LIN {X 0,Y 530.945,Z 338.971,A -85,B 0,C 180,E1 -4197.132,E2 -4197.132} C_VEL
LIN {X 0,Y 530.932,Z 338.967,A -85,B 0,C 180,E1 -4199.801,E2 -4199.801} C_VEL
LIN {X 0,Y 530.986,Z 339.128,A -85,B 0,C 180,E1 -4201.443,E2 -4201.443} C_VEL
LIN {X 0,Y 533.881,Z 351.837,A -85,B 0,C 180,E1 -4203.201,E2 -4203.201} C_VEL
LIN {X 0,Y 533.349,Z 375.523,A -85,B 0,C 180,E1 -4206.096,E2 -4206.096} C_VEL
LIN {X 0,Y 532.844,Z 398.324,A -85,B 0,C 180,E1 -4208.824,E2 -4208.824} C_VEL
LIN {X 0,Y 535.193,Z 410.616,A -85,B 0,C 180,E1 -4209.118,E2 -4209.118} C_VEL
LIN {X 0,Y 534.278,Z 564.153,A -85,B 0,C 180,E1 -4211.249,E2 -4211.249} C_VEL
LIN {X 0,Y 534.01,Z 579.764,A -85,B 0,C 180,E1 -4211.612,E2 -4211.612} C_VEL
LIN {X 0,Y 533.688,Z 594.764,A -85,B 0,C 180,E1 -4212.122,E2 -4212.122} C_VEL
LIN {X 0,Y 533.332,Z 608.76,A -85,B 0,C 180,E1 -4212.753,E2 -4212.753} C_VEL
LIN {X 0,Y 532.844,Z 622.489,A -85,B 0,C 180,E1 -4213.526,E2 -4213.526} C_VEL
LIN {X 0,Y 532.401,Z 636.442,A -85,B 0,C 180,E1 -4214.503,E2 -4214.503} C_VEL
LIN {X 0,Y 531.99,Z 647.758,A -85,B 0,C 180,E1 -4215.463,E2 -4215.463} C_VEL
LIN {X 0,Y 531.655,Z 657.488,A -85,B 0,C 180,E1 -4216.43,E2 -4216.43} C_VEL
LIN {X 0,Y 531.343,Z 665.917,A -85,B 0,C 180,E1 -4217.394,E2 -4217.394} C_VEL
LIN {X 0,Y 531.108,Z 672.885,A -85,B 0,C 180,E1 -4218.3,E2 -4218.3} C_VEL
LIN {X 0,Y 531.005,Z 679.757,A -85,B 0,C 180,E1 -4219.322,E2 -4219.322} C_VEL
LIN {X 0,Y 530.768,Z 686.452,A -85,B 0,C 180,E1 -4220.473,E2 -4220.473} C_VEL
LIN {X 0,Y 530.667,Z 692.162,A -85,B 0,C 180,E1 -4221.623,E2 -4221.623} C_VEL
LIN {X 0,Y 530.573,Z 696.984,A -85,B 0,C 180,E1 -4222.771,E2 -4222.771} C_VEL
LIN {X 0,Y 530.515,Z 701.005,A -85,B 0,C 180,E1 -4223.916,E2 -4223.916} C_VEL
LIN {X 0,Y 530.412,Z 705.143,A -85,B 0,C 180,E1 -4225.44,E2 -4225.44} C_VEL
LIN {X 0,Y 530.481,Z 706.833,A -85,B 0,C 180,E1 -4226.202,E2 -4226.202} C_VEL
LIN {X 0,Y 530.409,Z 709.125,A -85,B 0,C 180,E1 -4227.722,E2 -4227.722} C_VEL
LIN {X 0,Y 530.34,Z 710.269,A -85,B 0,C 180,E1 -4229.241,E2 -4229.241} C_VEL
LIN {X 0,Y 530.341,Z 710.497,A -85,B 0,C 180,E1 -4230,E2 -4230} C_VEL
LIN {X 0,Y 530.359,Z 709.942,A -85,B 0,C 180,E1 -4231.519,E2 -4231.519} C_VEL
LIN {X 0,Y 530.45,Z 708.224,A -85,B 0,C 180,E1 -4233.038,E2 -4233.038} C_VEL
LIN {X 0,Y 530.481,Z 706.999,A -85,B 0,C 180,E1 -4233.798,E2 -4233.798} C_VEL
LIN {X 0,Y 530.508,Z 703.526,A -85,B 0,C 180,E1 -4235.321,E2 -4235.321} C_VEL
LIN {X 0,Y 530.55,Z 698.716,A -85,B 0,C 180,E1 -4236.847,E2 -4236.847} C_VEL
LIN {X 0,Y 530.636,Z 694.25,A -85,B 0,C 180,E1 -4237.994,E2 -4237.994} C_VEL
LIN {X 0,Y 530.742,Z 688.921,A -85,B 0,C 180,E1 -4239.143,E2 -4239.143} C_VEL
LIN {X 0,Y 530.926,Z 682.638,A -85,B 0,C 180,E1 -4240.294,E2 -4240.294} C_VEL
LIN {X 0,Y 531.066,Z 675.267,A -85,B 0,C 180,E1 -4241.45,E2 -4241.45} C_VEL
LIN {X 0,Y 531.288,Z 668.195,A -85,B 0,C 180,E1 -4242.413,E2 -4242.413} C_VEL
LIN {X 0,Y 531.589,Z 660.096,A -85,B 0,C 180,E1 -4243.377,E2 -4243.377} C_VEL
LIN {X 0,Y 531.893,Z 650.752,A -85,B 0,C 180,E1 -4244.344,E2 -4244.344} C_VEL
LIN {X 0,Y 532.284,Z 639.846,A -85,B 0,C 180,E1 -4245.312,E2 -4245.312} C_VEL
LIN {X 0,Y 532.646,Z 628.232,A -85,B 0,C 180,E1 -4246.185,E2 -4246.185} C_VEL
LIN {X 0,Y 533.167,Z 614.163,A -85,B 0,C 180,E1 -4247.055,E2 -4247.055} C_VEL
LIN {X 0,Y 533.547,Z 600.41,A -85,B 0,C 180,E1 -4247.734,E2 -4247.734} C_VEL
LIN {X 0,Y 533.892,Z 585.818,A -85,B 0,C 180,E1 -4248.293,E2 -4248.293} C_VEL
LIN {X 0,Y 534.167,Z 571.375,A -85,B 0,C 180,E1 -4248.694,E2 -4248.694} C_VEL
LIN {X 0,Y 534.375,Z 554.599,A -85,B 0,C 180,E1 -4248.991,E2 -4248.991} C_VEL
LIN {X 0,Y 535.195,Z 410.641,A -85,B 0,C 180,E1 -4250.972,E2 -4250.972} C_VEL
LIN {X 0,Y 532.855,Z 398.387,A -85,B 0,C 180,E1 -4251.256,E2 -4251.256} C_VEL
LIN {X 0,Y 533.401,Z 372.991,A -85,B 0,C 180,E1 -4254.303,E2 -4254.303} C_VEL
LIN {X 0,Y 533.864,Z 352.576,A -85,B 0,C 180,E1 -4256.8,E2 -4256.8} C_VEL
LIN {X 0,Y 533.375,Z 349.148,A -85,B 0,C 180,E1 -4257.25,E2 -4257.25} C_VEL
LIN {X 0,Y 530.957,Z 339.096,A -85,B 0,C 180,E1 -4258.66,E2 -4258.66} C_VEL
LIN {X 0,Y 530.935,Z 338.972,A -85,B 0,C 180,E1 -4261.081,E2 -4261.081} C_VEL
LIN {X 0,Y 530.932,Z 338.973,A -85,B 0,C 180,E1 -4263.777,E2 -4263.777} C_VEL
LIN {X 0,Y 530.902,Z 338.976,A -85,B 0,C 180,E1 -4266.563,E2 -4266.563} C_VEL
LIN {X 0,Y 530.938,Z 338.971,A -85,B 0,C 180,E1 -4269.448,E2 -4269.448} C_VEL
LIN {X 0,Y 530.91,Z 338.974,A -85,B 0,C 180,E1 -4272.463,E2 -4272.463} C_VEL
LIN {X 0,Y 530.963,Z 338.969,A -85,B 0,C 180,E1 -4275.45,E2 -4275.45} C_VEL
LIN {X 0,Y 530.918,Z 338.973,A -85,B 0,C 180,E1 -4278.557,E2 -4278.557} C_VEL
LIN {X 0,Y 530.947,Z 338.972,A -85,B 0,C 180,E1 -4281.528,E2 -4281.528} C_VEL
LIN {X 0,Y 530.934,Z 338.969,A -85,B 0,C 180,E1 -4284.378,E2 -4284.378} C_VEL
LIN {X 0,Y 530.967,Z 338.967,A -85,B 0,C 180,E1 -4287.133,E2 -4287.133} C_VEL
LIN {X 0,Y 530.96,Z 338.975,A -85,B 0,C 180,E1 -4289.802,E2 -4289.802} C_VEL
LIN {X 0,Y 530.963,Z 338.963,A -85,B 0,C 180,E1 -4292.478,E2 -4292.478} C_VEL
LIN {X 0,Y 530.95,Z 338.968,A -85,B 0,C 180,E1 -4294.94,E2 -4294.94} C_VEL
LIN {X 0,Y 530.978,Z 338.967,A -85,B 0,C 180,E1 -4297.898,E2 -4297.898} C_VEL
LIN {X 0,Y 530.983,Z 338.964,A -85,B 0,C 180,E1 -4300.677,E2 -4300.677} C_VEL
LIN {X 0,Y 530.965,Z 338.965,A -85,B 0,C 180,E1 -4303.07,E2 -4303.07} C_VEL
LIN {X 0,Y 531.02,Z 338.965,A -85,B 0,C 180,E1 -4305.436,E2 -4305.436} C_VEL
LIN {X 0,Y 531.036,Z 338.953,A -85,B 0,C 180,E1 -4308.55,E2 -4308.55} C_VEL
LIN {X 0,Y 531.035,Z 338.965,A -85,B 0,C 180,E1 -4311.629,E2 -4311.629} C_VEL
LIN {X 0,Y 531.117,Z 338.943,A -85,B 0,C 180,E1 -4314.685,E2 -4314.685} C_VEL
LIN {X 0,Y 531.14,Z 338.949,A -85,B 0,C 180,E1 -4317.725,E2 -4317.725} C_VEL
LIN {X 0,Y 531.149,Z 338.941,A -85,B 0,C 180,E1 -4320.758,E2 -4320.758} C_VEL
LIN {X 0,Y 531.101,Z 338.949,A -85,B 0,C 180,E1 -4323.034,E2 -4323.034} C_VEL
LIN {X 0,Y 531.074,Z 338.951,A -85,B 0,C 180,E1 -4326.077,E2 -4326.077} C_VEL
LIN {X 0,Y 531.023,Z 338.96,A -85,B 0,C 180,E1 -4329.138,E2 -4329.138} C_VEL
LIN {X 0,Y 531.041,Z 338.954,A -85,B 0,C 180,E1 -4332.225,E2 -4332.225} C_VEL
LIN {X 0,Y 530.994,Z 338.968,A -85,B 0,C 180,E1 -4335.35,E2 -4335.35} C_VEL
LIN {X 0,Y 530.987,Z 338.962,A -85,B 0,C 180,E1 -4338.521,E2 -4338.521} C_VEL
LIN {X 0,Y 530.999,Z 338.963,A -85,B 0,C 180,E1 -4340.938,E2 -4340.938} C_VEL
LIN {X 0,Y 530.966,Z 338.963,A -85,B 0,C 180,E1 -4344.225,E2 -4344.225} C_VEL
LIN {X 0,Y 531.002,Z 338.963,A -85,B 0,C 180,E1 -4346.744,E2 -4346.744} C_VEL
LIN {X 0,Y 530.982,Z 338.966,A -85,B 0,C 180,E1 -4349.322,E2 -4349.322} C_VEL
LIN {X 0,Y 530.966,Z 338.966,A -85,B 0,C 180,E1 -4352.1,E2 -4352.1} C_VEL
LIN {X 0,Y 530.97,Z 338.968,A -85,B 0,C 180,E1 -4354.851,E2 -4354.851} C_VEL
LIN {X 0,Y 530.966,Z 338.967,A -85,B 0,C 180,E1 -4357.508,E2 -4357.508} C_VEL
LIN {X 0,Y 530.984,Z 338.952,A -85,B 0,C 180,E1 -4360.433,E2 -4360.433} C_VEL
LIN {X 0,Y 530.965,Z 338.969,A -85,B 0,C 180,E1 -4363.494,E2 -4363.494} C_VEL
LIN {X 0,Y 530.965,Z 338.963,A -85,B 0,C 180,E1 -4366.505,E2 -4366.505} C_VEL
LIN {X 0,Y 530.985,Z 338.965,A -85,B 0,C 180,E1 -4369.567,E2 -4369.567} C_VEL
LIN {X 0,Y 530.968,Z 338.971,A -85,B 0,C 180,E1 -4372.577,E2 -4372.577} C_VEL
LIN {X 0,Y 530.982,Z 338.969,A -85,B 0,C 180,E1 -4375.31,E2 -4375.31} C_VEL
LIN {X 0,Y 530.968,Z 338.967,A -85,B 0,C 180,E1 -4378.032,E2 -4378.032} C_VEL
LIN {X 0,Y 530.989,Z 338.971,A -85,B 0,C 180,E1 -4380.874,E2 -4380.874} C_VEL
LIN {X 0,Y 531.044,Z 339.142,A -85,B 0,C 180,E1 -4381.924,E2 -4381.924} C_VEL
LIN {X 0,Y 534.398,Z 352.329,A -85,B 0,C 180,E1 -4383.691,E2 -4383.691} C_VEL
LIN {X 0,Y 533.668,Z 375.374,A -85,B 0,C 180,E1 -4386.318,E2 -4386.318} C_VEL
LIN {X 0,Y 533.029,Z 397.899,A -85,B 0,C 180,E1 -4388.826,E2 -4388.826} C_VEL
LIN {X 0,Y 535.1,Z 409.701,A -85,B 0,C 180,E1 -4389.1,E2 -4389.1} C_VEL
LIN {X 0,Y 534.127,Z 564.616,A -85,B 0,C 180,E1 -4391.261,E2 -4391.261} C_VEL
LIN {X 0,Y 533.892,Z 580.328,A -85,B 0,C 180,E1 -4391.633,E2 -4391.633} C_VEL
LIN {X 0,Y 533.573,Z 594.596,A -85,B 0,C 180,E1 -4392.118,E2 -4392.118} C_VEL
LIN {X 0,Y 533.2,Z 608.743,A -85,B 0,C 180,E1 -4392.749,E2 -4392.749} C_VEL
LIN {X 0,Y 532.766,Z 622.554,A -85,B 0,C 180,E1 -4393.524,E2 -4393.524} C_VEL
LIN {X 0,Y 532.379,Z 635.728,A -85,B 0,C 180,E1 -4394.434,E2 -4394.434} C_VEL
LIN {X 0,Y 531.954,Z 648.089,A -85,B 0,C 180,E1 -4395.462,E2 -4395.462} C_VEL
LIN {X 0,Y 531.608,Z 659.731,A -85,B 0,C 180,E1 -4396.623,E2 -4396.623} C_VEL
LIN {X 0,Y 531.286,Z 669.388,A -85,B 0,C 180,E1 -4397.781,E2 -4397.781} C_VEL
LIN {X 0,Y 531.051,Z 678.853,A -85,B 0,C 180,E1 -4399.13,E2 -4399.13} C_VEL
LIN {X 0,Y 530.764,Z 686.735,A -85,B 0,C 180,E1 -4400.473,E2 -4400.473} C_VEL
LIN {X 0,Y 530.64,Z 694.089,A -85,B 0,C 180,E1 -4402.006,E2 -4402.006} C_VEL
LIN {X 0,Y 530.545,Z 699.699,A -85,B 0,C 180,E1 -4403.467,E2 -4403.467} C_VEL
LIN {X 0,Y 530.509,Z 703.386,A -85,B 0,C 180,E1 -4404.679,E2 -4404.679} C_VEL
LIN {X 0,Y 530.481,Z 706.887,A -85,B 0,C 180,E1 -4406.202,E2 -4406.202} C_VEL
LIN {X 0,Y 530.408,Z 709.189,A -85,B 0,C 180,E1 -4407.722,E2 -4407.722} C_VEL
LIN {X 0,Y 530.34,Z 710.348,A -85,B 0,C 180,E1 -4409.241,E2 -4409.241} C_VEL
LIN {X 0,Y 530.34,Z 710.347,A -85,B 0,C 180,E1 -4410.759,E2 -4410.759} C_VEL
LIN {X 0,Y 530.408,Z 709.185,A -85,B 0,C 180,E1 -4412.278,E2 -4412.278} C_VEL
LIN {X 0,Y 530.481,Z 706.882,A -85,B 0,C 180,E1 -4413.798,E2 -4413.798} C_VEL
LIN {X 0,Y 530.509,Z 703.386,A -85,B 0,C 180,E1 -4415.321,E2 -4415.321} C_VEL
LIN {X 0,Y 530.55,Z 698.609,A -85,B 0,C 180,E1 -4416.847,E2 -4416.847} C_VEL
LIN {X 0,Y 530.665,Z 692.419,A -85,B 0,C 180,E1 -4418.377,E2 -4418.377} C_VEL
LIN {X 0,Y 530.809,Z 684.641,A -85,B 0,C 180,E1 -4419.911,E2 -4419.911} C_VEL
LIN {X 0,Y 531.056,Z 676.365,A -85,B 0,C 180,E1 -4421.257,E2 -4421.257} C_VEL
LIN {X 0,Y 531.383,Z 666.39,A -85,B 0,C 180,E1 -4422.605,E2 -4422.605} C_VEL
LIN {X 0,Y 531.708,Z 656.119,A -85,B 0,C 180,E1 -4423.764,E2 -4423.764} C_VEL
LIN {X 0,Y 532.084,Z 643.687,A -85,B 0,C 180,E1 -4424.926,E2 -4424.926} C_VEL
LIN {X 0,Y 532.515,Z 631.406,A -85,B 0,C 180,E1 -4425.877,E2 -4425.877} C_VEL
LIN {X 0,Y 532.924,Z 617.492,A -85,B 0,C 180,E1 -4426.767,E2 -4426.767} C_VEL
LIN {X 0,Y 533.287,Z 603.31,A -85,B 0,C 180,E1 -4427.496,E2 -4427.496} C_VEL
LIN {X 0,Y 533.618,Z 588.738,A -85,B 0,C 180,E1 -4428.079,E2 -4428.079} C_VEL
LIN {X 0,Y 533.959,Z 573.588,A -85,B 0,C 180,E1 -4428.522,E2 -4428.522} C_VEL
LIN {X 0,Y 534.141,Z 557.458,A -85,B 0,C 180,E1 -4428.83,E2 -4428.83} C_VEL
LIN {X 0,Y 534.954,Z 409.306,A -85,B 0,C 180,E1 -4430.883,E2 -4430.883} C_VEL
LIN {X 0,Y 533.023,Z 398.201,A -85,B 0,C 180,E1 -4431.125,E2 -4431.125} C_VEL
LIN {X 0,Y 533.541,Z 376.812,A -85,B 0,C 180,E1 -4433.482,E2 -4433.482} C_VEL
LIN {X 0,Y 534.319,Z 352.2,A -85,B 0,C 180,E1 -4436.292,E2 -4436.292} C_VEL
LIN {X 0,Y 531.049,Z 339.118,A -85,B 0,C 180,E1 -4438.089,E2 -4438.089} C_VEL
LIN {X 0,Y 530.958,Z 338.975,A -85,B 0,C 180,E1 -4441.079,E2 -4441.079} C_VEL
LIN {X 0,Y 530.99,Z 338.965,A -85,B 0,C 180,E1 -4443.773,E2 -4443.773} C_VEL
LIN {X 0,Y 530.96,Z 338.974,A -85,B 0,C 180,E1 -4446.558,E2 -4446.558} C_VEL
LIN {X 0,Y 530.987,Z 338.967,A -85,B 0,C 180,E1 -4449.444,E2 -4449.444} C_VEL
LIN {X 0,Y 530.979,Z 338.971,A -85,B 0,C 180,E1 -4452.457,E2 -4452.457} C_VEL
LIN {X 0,Y 530.978,Z 338.967,A -85,B 0,C 180,E1 -4455.622,E2 -4455.622} C_VEL
LIN {X 0,Y 530.99,Z 338.972,A -85,B 0,C 180,E1 -4458.564,E2 -4458.564} C_VEL
LIN {X 0,Y 530.954,Z 338.97,A -85,B 0,C 180,E1 -4461.529,E2 -4461.529} C_VEL
LIN {X 0,Y 530.948,Z 338.977,A -85,B 0,C 180,E1 -4464.38,E2 -4464.38} C_VEL
LIN {X 0,Y 530.967,Z 338.97,A -85,B 0,C 180,E1 -4467.133,E2 -4467.133} C_VEL
LIN {X 0,Y 530.948,Z 338.975,A -85,B 0,C 180,E1 -4469.802,E2 -4469.802} C_VEL
LIN {X 0,Y 530.954,Z 338.976,A -85,B 0,C 180,E1 -4472.48,E2 -4472.48} C_VEL
LIN {X 0,Y 530.993,Z 339.163,A -85,B 0,C 180,E1 -4473.442,E2 -4473.442} C_VEL
LIN {X 0,Y 533.281,Z 349.071,A -85,B 0,C 180,E1 -4475.057,E2 -4475.057} C_VEL
LIN {X 0,Y 533.456,Z 353.457,A -85,B 0,C 180,E1 -4475.699,E2 -4475.699} C_VEL
LIN {X 0,Y 532.723,Z 376.404,A -85,B 0,C 180,E1 -4478.931,E2 -4478.931} C_VEL
LIN {X 0,Y 532.137,Z 397.45,A -85,B 0,C 180,E1 -4481.828,E2 -4481.828} C_VEL
LIN {X 0,Y 533.286,Z 403.741,A -85,B 0,C 180,E1 -4482.001,E2 -4482.001} C_VEL
LIN {X 0,Y 534.066,Z 408.919,A -85,B 0,C 180,E1 -4482.11,E2 -4482.11} C_VEL
LIN {X 0,Y 533.219,Z 536.961,A -85,B 0,C 180,E1 -4483.949,E2 -4483.949} C_VEL
LIN {X 0,Y 532.942,Z 551.427,A -85,B 0,C 180,E1 -4484.314,E2 -4484.314} C_VEL
LIN {X 0,Y 532.714,Z 565.736,A -85,B 0,C 180,E1 -4484.848,E2 -4484.848} C_VEL
LIN {X 0,Y 532.412,Z 578.426,A -85,B 0,C 180,E1 -4485.475,E2 -4485.475} C_VEL
LIN {X 0,Y 532.053,Z 590.85,A -85,B 0,C 180,E1 -4486.245,E2 -4486.245} C_VEL
LIN {X 0,Y 531.733,Z 602.123,A -85,B 0,C 180,E1 -4487.112,E2 -4487.112} C_VEL
LIN {X 0,Y 531.422,Z 613.157,A -85,B 0,C 180,E1 -4488.138,E2 -4488.138} C_VEL
LIN {X 0,Y 531.208,Z 622,A -85,B 0,C 180,E1 -4489.133,E2 -4489.133} C_VEL
LIN {X 0,Y 530.929,Z 630.682,A -85,B 0,C 180,E1 -4490.284,E2 -4490.284} C_VEL
LIN {X 0,Y 530.743,Z 638.877,A -85,B 0,C 180,E1 -4491.625,E2 -4491.625} C_VEL
LIN {X 0,Y 530.587,Z 644.644,A -85,B 0,C 180,E1 -4492.771,E2 -4492.771} C_VEL
LIN {X 0,Y 530.566,Z 650.752,A -85,B 0,C 180,E1 -4494.299,E2 -4494.299} C_VEL
LIN {X 0,Y 530.449,Z 654.284,A -85,B 0,C 180,E1 -4495.441,E2 -4495.441} C_VEL
LIN {X 0,Y 530.453,Z 657.771,A -85,B 0,C 180,E1 -4496.962,E2 -4496.962} C_VEL
LIN {X 0,Y 530.359,Z 659.74,A -85,B 0,C 180,E1 -4498.481,E2 -4498.481} C_VEL
LIN {X 0,Y 530.342,Z 660.496,A -85,B 0,C 180,E1 -4500,E2 -4500} C_VEL
LIN {X 0,Y 530.357,Z 659.816,A -85,B 0,C 180,E1 -4501.519,E2 -4501.519} C_VEL
LIN {X 0,Y 530.452,Z 657.919,A -85,B 0,C 180,E1 -4503.038,E2 -4503.038} C_VEL
LIN {X 0,Y 530.448,Z 654.528,A -85,B 0,C 180,E1 -4504.56,E2 -4504.56} C_VEL
LIN {X 0,Y 530.568,Z 649.767,A -85,B 0,C 180,E1 -4506.083,E2 -4506.083} C_VEL
LIN {X 0,Y 530.64,Z 643.271,A -85,B 0,C 180,E1 -4507.611,E2 -4507.611} C_VEL
LIN {X 0,Y 530.809,Z 636.09,A -85,B 0,C 180,E1 -4508.95,E2 -4508.95} C_VEL
LIN {X 0,Y 530.982,Z 628.546,A -85,B 0,C 180,E1 -4510.101,E2 -4510.101} C_VEL
LIN {X 0,Y 531.274,Z 619.564,A -85,B 0,C 180,E1 -4511.252,E2 -4511.252} C_VEL
LIN {X 0,Y 531.459,Z 610.473,A -85,B 0,C 180,E1 -4512.215,E2 -4512.215} C_VEL
LIN {X 0,Y 531.82,Z 599.737,A -85,B 0,C 180,E1 -4513.177,E2 -4513.177} C_VEL
LIN {X 0,Y 532.121,Z 587.852,A -85,B 0,C 180,E1 -4514.045,E2 -4514.045} C_VEL
LIN {X 0,Y 532.518,Z 574.763,A -85,B 0,C 180,E1 -4514.815,E2 -4514.815} C_VEL
LIN {X 0,Y 532.84,Z 562.962,A -85,B 0,C 180,E1 -4515.36,E2 -4515.36} C_VEL
LIN {X 0,Y 533.045,Z 549.361,A -85,B 0,C 180,E1 -4515.839,E2 -4515.839} C_VEL
LIN {X 0,Y 533.237,Z 536.026,A -85,B 0,C 180,E1 -4516.166,E2 -4516.166} C_VEL
LIN {X 0,Y 533.921,Z 407.703,A -85,B 0,C 180,E1 -4517.973,E2 -4517.973} C_VEL
LIN {X 0,Y 532.113,Z 397.871,A -85,B 0,C 180,E1 -4518.204,E2 -4518.204} C_VEL
LIN {X 0,Y 532.073,Z 396.512,A -85,B 0,C 180,E1 -4518.329,E2 -4518.329} C_VEL
LIN {X 0,Y 532.671,Z 373.671,A -85,B 0,C 180,E1 -4521.477,E2 -4521.477} C_VEL
LIN {X 0,Y 533.099,Z 360.019,A -85,B 0,C 180,E1 -4523.384,E2 -4523.384} C_VEL
LIN {X 0,Y 532.535,Z 356.591,A -85,B 0,C 180,E1 -4523.898,E2 -4523.898} C_VEL
LIN {X 0,Y 530.909,Z 353.505,A -85,B 0,C 180,E1 -4524.419,E2 -4524.419} C_VEL
LIN {X 0,Y 525.491,Z 345.703,A -85,B 0,C 180,E1 -4525.83,E2 -4525.83} C_VEL
LIN {X 0,Y 524.749,Z 343.526,A -85,B 0,C 180,E1 -4526.19,E2 -4526.19} C_VEL
LIN {X 0,Y 523.916,Z 339.972,A -85,B 0,C 180,E1 -4526.812,E2 -4526.812} C_VEL
LIN {X 0,Y 523.868,Z 339.856,A -85,B 0,C 180,E1 -4529.761,E2 -4529.761} C_VEL
LIN {X 0,Y 523.896,Z 339.852,A -85,B 0,C 180,E1 -4532.452,E2 -4532.452} C_VEL
LIN {X 0,Y 523.882,Z 339.85,A -85,B 0,C 180,E1 -4535.23,E2 -4535.23} C_VEL
LIN {X 0,Y 523.888,Z 339.856,A -85,B 0,C 180,E1 -4538.104,E2 -4538.104} C_VEL
LIN {X 0,Y 523.876,Z 339.849,A -85,B 0,C 180,E1 -4541.3,E2 -4541.3} C_VEL
LIN {X 0,Y 523.93,Z 339.845,A -85,B 0,C 180,E1 -4544.688,E2 -4544.688} C_VEL
LIN {X 0,Y 523.886,Z 339.85,A -85,B 0,C 180,E1 -4547.874,E2 -4547.874} C_VEL
LIN {X 0,Y 523.894,Z 339.846,A -85,B 0,C 180,E1 -4551.084,E2 -4551.084} C_VEL
LIN {X 0,Y 523.853,Z 339.855,A -85,B 0,C 180,E1 -4553.821,E2 -4553.821} C_VEL
LIN {X 0,Y 523.896,Z 339.851,A -85,B 0,C 180,E1 -4556.632,E2 -4556.632} C_VEL
LIN {X 0,Y 523.908,Z 339.847,A -85,B 0,C 180,E1 -4559.352,E2 -4559.352} C_VEL
LIN {X 0,Y 523.953,Z 340.098,A -85,B 0,C 180,E1 -4561.208,E2 -4561.208} C_VEL
LIN {X 0,Y 527.02,Z 353.216,A -85,B 0,C 180,E1 -4563.038,E2 -4563.038} C_VEL
LIN {X 0,Y 526.614,Z 372.459,A -85,B 0,C 180,E1 -4565.425,E2 -4565.425} C_VEL
LIN {X 0,Y 526.029,Z 398.344,A -85,B 0,C 180,E1 -4568.546,E2 -4568.546} C_VEL
LIN {X 0,Y 528.57,Z 411.924,A -85,B 0,C 180,E1 -4568.864,E2 -4568.864} C_VEL
LIN {X 0,Y 527.559,Z 564.979,A -85,B 0,C 180,E1 -4571.018,E2 -4571.018} C_VEL
LIN {X 0,Y 527.254,Z 580.553,A -85,B 0,C 180,E1 -4571.393,E2 -4571.393} C_VEL
LIN {X 0,Y 526.913,Z 594.711,A -85,B 0,C 180,E1 -4571.884,E2 -4571.884} C_VEL
LIN {X 0,Y 526.533,Z 608.749,A -85,B 0,C 180,E1 -4572.523,E2 -4572.523} C_VEL
LIN {X 0,Y 526,Z 622.447,A -85,B 0,C 180,E1 -4573.306,E2 -4573.306} C_VEL
LIN {X 0,Y 525.548,Z 635.473,A -85,B 0,C 180,E1 -4574.223,E2 -4574.223} C_VEL
LIN {X 0,Y 525.063,Z 647.759,A -85,B 0,C 180,E1 -4575.267,E2 -4575.267} C_VEL
LIN {X 0,Y 524.631,Z 659.31,A -85,B 0,C 180,E1 -4576.442,E2 -4576.442} C_VEL
LIN {X 0,Y 524.227,Z 670.524,A -85,B 0,C 180,E1 -4577.81,E2 -4577.81} C_VEL
LIN {X 0,Y 523.988,Z 679.779,A -85,B 0,C 180,E1 -4579.177,E2 -4579.177} C_VEL
LIN {X 0,Y 523.701,Z 686.457,A -85,B 0,C 180,E1 -4580.343,E2 -4580.343} C_VEL
LIN {X 0,Y 523.614,Z 692.158,A -85,B 0,C 180,E1 -4581.51,E2 -4581.51} C_VEL
LIN {X 0,Y 523.487,Z 696.981,A -85,B 0,C 180,E1 -4582.672,E2 -4582.672} C_VEL
LIN {X 0,Y 523.422,Z 701,A -85,B 0,C 180,E1 -4583.834,E2 -4583.834} C_VEL
LIN {X 0,Y 523.441,Z 703.255,A -85,B 0,C 180,E1 -4584.607,E2 -4584.607} C_VEL
LIN {X 0,Y 523.402,Z 706.837,A -85,B 0,C 180,E1 -4586.15,E2 -4586.15} C_VEL
LIN {X 0,Y 523.332,Z 709.121,A -85,B 0,C 180,E1 -4587.691,E2 -4587.691} C_VEL
LIN {X 0,Y 523.246,Z 710.263,A -85,B 0,C 180,E1 -4589.23,E2 -4589.23} C_VEL
LIN {X 0,Y 523.244,Z 710.497,A -85,B 0,C 180,E1 -4590,E2 -4590} C_VEL
LIN {X 0,Y 523.273,Z 709.936,A -85,B 0,C 180,E1 -4591.539,E2 -4591.539} C_VEL
LIN {X 0,Y 523.359,Z 708.217,A -85,B 0,C 180,E1 -4593.079,E2 -4593.079} C_VEL
LIN {X 0,Y 523.403,Z 706.992,A -85,B 0,C 180,E1 -4593.85,E2 -4593.85} C_VEL
LIN {X 0,Y 523.44,Z 703.519,A -85,B 0,C 180,E1 -4595.393,E2 -4595.393} C_VEL
LIN {X 0,Y 523.481,Z 698.708,A -85,B 0,C 180,E1 -4596.94,E2 -4596.94} C_VEL
LIN {X 0,Y 523.56,Z 694.24,A -85,B 0,C 180,E1 -4598.103,E2 -4598.103} C_VEL
LIN {X 0,Y 523.666,Z 688.917,A -85,B 0,C 180,E1 -4599.268,E2 -4599.268} C_VEL
LIN {X 0,Y 523.903,Z 682.646,A -85,B 0,C 180,E1 -4600.434,E2 -4600.434} C_VEL
LIN {X 0,Y 524.05,Z 675.285,A -85,B 0,C 180,E1 -4601.605,E2 -4601.605} C_VEL
LIN {X 0,Y 524.359,Z 666.68,A -85,B 0,C 180,E1 -4602.777,E2 -4602.777} C_VEL
LIN {X 0,Y 524.761,Z 656.574,A -85,B 0,C 180,E1 -4603.95,E2 -4603.95} C_VEL
LIN {X 0,Y 525.237,Z 644.564,A -85,B 0,C 180,E1 -4605.116,E2 -4605.116} C_VEL
LIN {X 0,Y 525.678,Z 632.372,A -85,B 0,C 180,E1 -4606.106,E2 -4606.106} C_VEL
LIN {X 0,Y 526.168,Z 619.201,A -85,B 0,C 180,E1 -4606.989,E2 -4606.989} C_VEL
LIN {X 0,Y 526.584,Z 604.649,A -85,B 0,C 180,E1 -4607.776,E2 -4607.776} C_VEL
LIN {X 0,Y 527.018,Z 590.741,A -85,B 0,C 180,E1 -4608.364,E2 -4608.364} C_VEL
LIN {X 0,Y 527.379,Z 574.818,A -85,B 0,C 180,E1 -4608.857,E2 -4608.857} C_VEL
LIN {X 0,Y 527.629,Z 560.181,A -85,B 0,C 180,E1 -4609.158,E2 -4609.158} C_VEL
LIN {X 0,Y 528.521,Z 411.529,A -85,B 0,C 180,E1 -4611.234,E2 -4611.234} C_VEL
LIN {X 0,Y 526.007,Z 398.337,A -85,B 0,C 180,E1 -4611.541,E2 -4611.541} C_VEL
LIN {X 0,Y 526.584,Z 373.207,A -85,B 0,C 180,E1 -4614.573,E2 -4614.573} C_VEL
LIN {X 0,Y 527.053,Z 353.953,A -85,B 0,C 180,E1 -4616.96,E2 -4616.96} C_VEL
LIN {X 0,Y 525.431,Z 346.223,A -85,B 0,C 180,E1 -4618.018,E2 -4618.018} C_VEL
LIN {X 0,Y 523.918,Z 339.938,A -85,B 0,C 180,E1 -4618.931,E2 -4618.931} C_VEL
LIN {X 0,Y 523.904,Z 339.848,A -85,B 0,C 180,E1 -4621.545,E2 -4621.545} C_VEL
LIN {X 0,Y 523.902,Z 339.853,A -85,B 0,C 180,E1 -4624.292,E2 -4624.292} C_VEL
LIN {X 0,Y 523.871,Z 339.856,A -85,B 0,C 180,E1 -4627.672,E2 -4627.672} C_VEL
LIN {X 0,Y 523.881,Z 339.852,A -85,B 0,C 180,E1 -4630.122,E2 -4630.122} C_VEL
LIN {X 0,Y 523.879,Z 339.849,A -85,B 0,C 180,E1 -4633.171,E2 -4633.171} C_VEL
LIN {X 0,Y 523.918,Z 339.851,A -85,B 0,C 180,E1 -4635.77,E2 -4635.77} C_VEL
LIN {X 0,Y 523.877,Z 339.85,A -85,B 0,C 180,E1 -4638.902,E2 -4638.902} C_VEL
LIN {X 0,Y 523.901,Z 339.854,A -85,B 0,C 180,E1 -4641.897,E2 -4641.897} C_VEL
LIN {X 0,Y 523.915,Z 339.842,A -85,B 0,C 180,E1 -4644.913,E2 -4644.913} C_VEL
LIN {X 0,Y 523.935,Z 339.847,A -85,B 0,C 180,E1 -4647.68,E2 -4647.68} C_VEL
LIN {X 0,Y 523.953,Z 339.84,A -85,B 0,C 180,E1 -4650.677,E2 -4650.677} C_VEL
LIN {X 0,Y 523.899,Z 339.851,A -85,B 0,C 180,E1 -4653.724,E2 -4653.724} C_VEL
LIN {X 0,Y 523.91,Z 339.845,A -85,B 0,C 180,E1 -4656.269,E2 -4656.269} C_VEL
LIN {X 0,Y 523.946,Z 339.837,A -85,B 0,C 180,E1 -4658.767,E2 -4658.767} C_VEL
LIN {X 0,Y 523.938,Z 339.845,A -85,B 0,C 180,E1 -4661.22,E2 -4661.22} C_VEL
LIN {X 0,Y 523.923,Z 339.846,A -85,B 0,C 180,E1 -4663.638,E2 -4663.638} C_VEL
LIN {X 0,Y 523.935,Z 339.844,A -85,B 0,C 180,E1 -4666.028,E2 -4666.028} C_VEL
LIN {X 0,Y 523.993,Z 339.834,A -85,B 0,C 180,E1 -4669.177,E2 -4669.177} C_VEL
LIN {X 0,Y 524.006,Z 339.833,A -85,B 0,C 180,E1 -4672.292,E2 -4672.292} C_VEL
LIN {X 0,Y 524.078,Z 339.819,A -85,B 0,C 180,E1 -4674.614,E2 -4674.614} C_VEL
LIN {X 0,Y 524.111,Z 339.825,A -85,B 0,C 180,E1 -4677.694,E2 -4677.694} C_VEL
LIN {X 0,Y 524.12,Z 339.816,A -85,B 0,C 180,E1 -4680.768,E2 -4680.768} C_VEL
LIN {X 0,Y 524.042,Z 339.829,A -85,B 0,C 180,E1 -4683.075,E2 -4683.075} C_VEL
LIN {X 0,Y 524.033,Z 339.827,A -85,B 0,C 180,E1 -4686.159,E2 -4686.159} C_VEL
LIN {X 0,Y 523.993,Z 339.837,A -85,B 0,C 180,E1 -4689.262,E2 -4689.262} C_VEL
LIN {X 0,Y 524.004,Z 339.834,A -85,B 0,C 180,E1 -4691.739,E2 -4691.739} C_VEL
LIN {X 0,Y 523.993,Z 339.835,A -85,B 0,C 180,E1 -4695.052,E2 -4695.052} C_VEL
LIN {X 0,Y 523.948,Z 339.839,A -85,B 0,C 180,E1 -4697.969,E2 -4697.969} C_VEL
LIN {X 0,Y 523.973,Z 339.833,A -85,B 0,C 180,E1 -4700.41,E2 -4700.41} C_VEL
LIN {X 0,Y 523.911,Z 339.849,A -85,B 0,C 180,E1 -4702.893,E2 -4702.893} C_VEL
LIN {X 0,Y 523.985,Z 339.834,A -85,B 0,C 180,E1 -4706.02,E2 -4706.02} C_VEL
LIN {X 0,Y 523.94,Z 339.846,A -85,B 0,C 180,E1 -4708.875,E2 -4708.875} C_VEL
LIN {X 0,Y 523.921,Z 339.847,A -85,B 0,C 180,E1 -4711.544,E2 -4711.544} C_VEL
LIN {X 0,Y 523.933,Z 339.839,A -85,B 0,C 180,E1 -4714.29,E2 -4714.29} C_VEL
LIN {X 0,Y 523.908,Z 339.851,A -85,B 0,C 180,E1 -4717.132,E2 -4717.132} C_VEL
LIN {X 0,Y 523.937,Z 339.827,A -85,B 0,C 180,E1 -4720.13,E2 -4720.13} C_VEL
LIN {X 0,Y 523.938,Z 339.84,A -85,B 0,C 180,E1 -4722.459,E2 -4722.459} C_VEL
LIN {X 0,Y 523.956,Z 339.837,A -85,B 0,C 180,E1 -4725.309,E2 -4725.309} C_VEL
LIN {X 0,Y 523.962,Z 339.841,A -85,B 0,C 180,E1 -4728.689,E2 -4728.689} C_VEL
LIN {X 0,Y 523.917,Z 339.845,A -85,B 0,C 180,E1 -4731.898,E2 -4731.898} C_VEL
LIN {X 0,Y 523.925,Z 339.85,A -85,B 0,C 180,E1 -4734.911,E2 -4734.911} C_VEL
LIN {X 0,Y 523.936,Z 339.844,A -85,B 0,C 180,E1 -4737.68,E2 -4737.68} C_VEL
LIN {X 0,Y 523.955,Z 339.846,A -85,B 0,C 180,E1 -4740.676,E2 -4740.676} C_VEL
LIN {X 0,Y 523.98,Z 339.999,A -85,B 0,C 180,E1 -4741.62,E2 -4741.62} C_VEL
LIN {X 0,Y 527.524,Z 353.673,A -85,B 0,C 180,E1 -4743.493,E2 -4743.493} C_VEL
LIN {X 0,Y 527.164,Z 368.063,A -85,B 0,C 180,E1 -4745.172,E2 -4745.172} C_VEL
LIN {X 0,Y 526.248,Z 396.2,A -85,B 0,C 180,E1 -4748.381,E2 -4748.381} C_VEL
LIN {X 0,Y 526.265,Z 398.528,A -85,B 0,C 180,E1 -4748.586,E2 -4748.586} C_VEL
LIN {X 0,Y 528.408,Z 410.584,A -85,B 0,C 180,E1 -4748.853,E2 -4748.853} C_VEL
LIN {X 0,Y 527.299,Z 564.913,A -85,B 0,C 180,E1 -4751.054,E2 -4751.054} C_VEL
LIN {X 0,Y 527.048,Z 580.608,A -85,B 0,C 180,E1 -4751.436,E2 -4751.436} C_VEL
LIN {X 0,Y 526.687,Z 595.966,A -85,B 0,C 180,E1 -4751.976,E2 -4751.976} C_VEL
LIN {X 0,Y 526.278,Z 609.805,A -85,B 0,C 180,E1 -4752.615,E2 -4752.615} C_VEL
LIN {X 0,Y 525.821,Z 623.364,A -85,B 0,C 180,E1 -4753.4,E2 -4753.4} C_VEL
LIN {X 0,Y 525.386,Z 637.273,A -85,B 0,C 180,E1 -4754.393,E2 -4754.393} C_VEL
LIN {X 0,Y 524.905,Z 649.626,A -85,B 0,C 180,E1 -4755.461,E2 -4755.461} C_VEL
LIN {X 0,Y 524.54,Z 660.991,A -85,B 0,C 180,E1 -4756.637,E2 -4756.637} C_VEL
LIN {X 0,Y 524.137,Z 672.004,A -85,B 0,C 180,E1 -4758.005,E2 -4758.005} C_VEL
LIN {X 0,Y 523.926,Z 681.152,A -85,B 0,C 180,E1 -4759.371,E2 -4759.371} C_VEL
LIN {X 0,Y 523.699,Z 688.723,A -85,B 0,C 180,E1 -4760.733,E2 -4760.733} C_VEL
LIN {X 0,Y 523.535,Z 695.7,A -85,B 0,C 180,E1 -4762.285,E2 -4762.285} C_VEL
LIN {X 0,Y 523.44,Z 701.162,A -85,B 0,C 180,E1 -4763.834,E2 -4763.834} C_VEL
LIN {X 0,Y 523.323,Z 705.29,A -85,B 0,C 180,E1 -4765.378,E2 -4765.378} C_VEL
LIN {X 0,Y 523.358,Z 708.183,A -85,B 0,C 180,E1 -4766.921,E2 -4766.921} C_VEL
LIN {X 0,Y 523.272,Z 709.909,A -85,B 0,C 180,E1 -4768.461,E2 -4768.461} C_VEL
LIN {X 0,Y 523.243,Z 710.5,A -85,B 0,C 180,E1 -4770,E2 -4770} C_VEL
LIN {X 0,Y 523.272,Z 709.906,A -85,B 0,C 180,E1 -4771.539,E2 -4771.539} C_VEL
LIN {X 0,Y 523.358,Z 708.178,A -85,B 0,C 180,E1 -4773.079,E2 -4773.079} C_VEL
LIN {X 0,Y 523.323,Z 705.287,A -85,B 0,C 180,E1 -4774.622,E2 -4774.622} C_VEL
LIN {X 0,Y 523.427,Z 701.165,A -85,B 0,C 180,E1 -4776.166,E2 -4776.166} C_VEL
LIN {X 0,Y 523.535,Z 695.7,A -85,B 0,C 180,E1 -4777.715,E2 -4777.715} C_VEL
LIN {X 0,Y 523.699,Z 688.716,A -85,B 0,C 180,E1 -4779.267,E2 -4779.267} C_VEL
LIN {X 0,Y 523.925,Z 681.127,A -85,B 0,C 180,E1 -4780.629,E2 -4780.629} C_VEL
LIN {X 0,Y 524.151,Z 671.894,A -85,B 0,C 180,E1 -4782.002,E2 -4782.002} C_VEL
LIN {X 0,Y 524.54,Z 660.869,A -85,B 0,C 180,E1 -4783.363,E2 -4783.363} C_VEL
LIN {X 0,Y 524.851,Z 649.425,A -85,B 0,C 180,E1 -4784.541,E2 -4784.541} C_VEL
LIN {X 0,Y 525.339,Z 637.221,A -85,B 0,C 180,E1 -4785.588,E2 -4785.588} C_VEL
LIN {X 0,Y 525.736,Z 624.405,A -85,B 0,C 180,E1 -4786.503,E2 -4786.503} C_VEL
LIN {X 0,Y 526.209,Z 610.979,A -85,B 0,C 180,E1 -4787.288,E2 -4787.288} C_VEL
LIN {X 0,Y 526.563,Z 597.37,A -85,B 0,C 180,E1 -4787.928,E2 -4787.928} C_VEL
LIN {X 0,Y 526.892,Z 583.172,A -85,B 0,C 180,E1 -4788.444,E2 -4788.444} C_VEL
LIN {X 0,Y 527.15,Z 567.861,A -85,B 0,C 180,E1 -4788.843,E2 -4788.843} C_VEL
LIN {X 0,Y 527.341,Z 546.344,A -85,B 0,C 180,E1 -4789.184,E2 -4789.184} C_VEL
LIN {X 0,Y 528.278,Z 412.875,A -85,B 0,C 180,E1 -4791.077,E2 -4791.077} C_VEL
LIN {X 0,Y 527.829,Z 408.072,A -85,B 0,C 180,E1 -4791.165,E2 -4791.165} C_VEL
LIN {X 0,Y 526.146,Z 398.194,A -85,B 0,C 180,E1 -4791.384,E2 -4791.384} C_VEL
LIN {X 0,Y 526.891,Z 373.007,A -85,B 0,C 180,E1 -4794.215,E2 -4794.215} C_VEL
LIN {X 0,Y 527.583,Z 354.589,A -85,B 0,C 180,E1 -4796.366,E2 -4796.366} C_VEL
LIN {X 0,Y 524.818,Z 343.023,A -85,B 0,C 180,E1 -4797.95,E2 -4797.95} C_VEL
LIN {X 0,Y 523.986,Z 339.959,A -85,B 0,C 180,E1 -4798.434,E2 -4798.434} C_VEL
LIN {X 0,Y 523.922,Z 339.849,A -85,B 0,C 180,E1 -4801.544,E2 -4801.544} C_VEL
LIN {X 0,Y 523.942,Z 339.844,A -85,B 0,C 180,E1 -4804.29,E2 -4804.29} C_VEL
LIN {X 0,Y 523.91,Z 339.852,A -85,B 0,C 180,E1 -4807.132,E2 -4807.132} C_VEL
LIN {X 0,Y 523.939,Z 339.845,A -85,B 0,C 180,E1 -4810.13,E2 -4810.13} C_VEL
LIN {X 0,Y 523.936,Z 339.849,A -85,B 0,C 180,E1 -4812.459,E2 -4812.459} C_VEL
LIN {X 0,Y 523.944,Z 339.844,A -85,B 0,C 180,E1 -4815.31,E2 -4815.31} C_VEL
LIN {X 0,Y 523.954,Z 339.847,A -85,B 0,C 180,E1 -4818.69,E2 -4818.69} C_VEL
LIN {X 0,Y 523.916,Z 339.848,A -85,B 0,C 180,E1 -4821.081,E2 -4821.081} C_VEL
LIN {X 0,Y 523.895,Z 339.851,A -85,B 0,C 180,E1 -4823.825,E2 -4823.825} C_VEL
LIN {X 0,Y 523.927,Z 339.85,A -85,B 0,C 180,E1 -4826.635,E2 -4826.635} C_VEL
LIN {X 0,Y 523.943,Z 339.845,A -85,B 0,C 180,E1 -4829.355,E2 -4829.355} C_VEL
LIN {X 0,Y 523.911,Z 339.853,A -85,B 0,C 180,E1 -4832.296,E2 -4832.296} C_VEL
LIN {X 0,Y 523.953,Z 340.143,A -85,B 0,C 180,E1 -4833.15,E2 -4833.15} C_VEL
LIN {X 0,Y 526.577,Z 351.389,A -85,B 0,C 180,E1 -4835.011,E2 -4835.011} C_VEL
LIN {X 0,Y 526.674,Z 355.098,A -85,B 0,C 180,E1 -4835.565,E2 -4835.565} C_VEL
LIN {X 0,Y 525.843,Z 378.059,A -85,B 0,C 180,E1 -4838.847,E2 -4838.847} C_VEL
LIN {X 0,Y 525.258,Z 397.604,A -85,B 0,C 180,E1 -4841.565,E2 -4841.565} C_VEL
LIN {X 0,Y 527.375,Z 409.252,A -85,B 0,C 180,E1 -4841.855,E2 -4841.855} C_VEL
LIN {X 0,Y 526.362,Z 537.283,A -85,B 0,C 180,E1 -4843.755,E2 -4843.755} C_VEL
LIN {X 0,Y 526.072,Z 552.083,A -85,B 0,C 180,E1 -4844.138,E2 -4844.138} C_VEL
LIN {X 0,Y 525.857,Z 565.53,A -85,B 0,C 180,E1 -4844.646,E2 -4844.646} C_VEL
LIN {X 0,Y 525.52,Z 578.354,A -85,B 0,C 180,E1 -4845.28,E2 -4845.28} C_VEL
LIN {X 0,Y 525.131,Z 590.867,A -85,B 0,C 180,E1 -4846.06,E2 -4846.06} C_VEL
LIN {X 0,Y 524.812,Z 602.202,A -85,B 0,C 180,E1 -4846.94,E2 -4846.94} C_VEL
LIN {X 0,Y 524.448,Z 612.897,A -85,B 0,C 180,E1 -4847.934,E2 -4847.934} C_VEL
LIN {X 0,Y 524.217,Z 622.195,A -85,B 0,C 180,E1 -4848.986,E2 -4848.986} C_VEL
LIN {X 0,Y 523.899,Z 630.892,A -85,B 0,C 180,E1 -4850.152,E2 -4850.152} C_VEL
LIN {X 0,Y 523.695,Z 639.112,A -85,B 0,C 180,E1 -4851.511,E2 -4851.511} C_VEL
LIN {X 0,Y 523.515,Z 646.615,A -85,B 0,C 180,E1 -4853.061,E2 -4853.061} C_VEL
LIN {X 0,Y 523.501,Z 650.991,A -85,B 0,C 180,E1 -4854.221,E2 -4854.221} C_VEL
LIN {X 0,Y 523.358,Z 654.494,A -85,B 0,C 180,E1 -4855.379,E2 -4855.379} C_VEL
LIN {X 0,Y 523.363,Z 657.938,A -85,B 0,C 180,E1 -4856.921,E2 -4856.921} C_VEL
LIN {X 0,Y 523.273,Z 659.891,A -85,B 0,C 180,E1 -4858.461,E2 -4858.461} C_VEL
LIN {X 0,Y 523.245,Z 660.634,A -85,B 0,C 180,E1 -4860,E2 -4860} C_VEL
LIN {X 0,Y 523.271,Z 659.959,A -85,B 0,C 180,E1 -4861.539,E2 -4861.539} C_VEL
LIN {X 0,Y 523.362,Z 658.072,A -85,B 0,C 180,E1 -4863.079,E2 -4863.079} C_VEL
LIN {X 0,Y 523.356,Z 654.711,A -85,B 0,C 180,E1 -4864.622,E2 -4864.622} C_VEL
LIN {X 0,Y 523.495,Z 649.961,A -85,B 0,C 180,E1 -4866.166,E2 -4866.166} C_VEL
LIN {X 0,Y 523.539,Z 645.257,A -85,B 0,C 180,E1 -4867.327,E2 -4867.327} C_VEL
LIN {X 0,Y 523.733,Z 638.509,A -85,B 0,C 180,E1 -4868.683,E2 -4868.683} C_VEL
LIN {X 0,Y 523.896,Z 630.071,A -85,B 0,C 180,E1 -4870.043,E2 -4870.043} C_VEL
LIN {X 0,Y 524.226,Z 621.305,A -85,B 0,C 180,E1 -4871.209,E2 -4871.209} C_VEL
LIN {X 0,Y 524.506,Z 610.553,A -85,B 0,C 180,E1 -4872.38,E2 -4872.38} C_VEL
LIN {X 0,Y 524.89,Z 599.751,A -85,B 0,C 180,E1 -4873.354,E2 -4873.354} C_VEL
LIN {X 0,Y 525.222,Z 587.826,A -85,B 0,C 180,E1 -4874.234,E2 -4874.234} C_VEL
LIN {X 0,Y 525.627,Z 574.654,A -85,B 0,C 180,E1 -4875.014,E2 -4875.014} C_VEL
LIN {X 0,Y 526.029,Z 561.14,A -85,B 0,C 180,E1 -4875.633,E2 -4875.633} C_VEL
LIN {X 0,Y 526.242,Z 547.557,A -85,B 0,C 180,E1 -4876.095,E2 -4876.095} C_VEL
LIN {X 0,Y 526.412,Z 532.5,A -85,B 0,C 180,E1 -4876.432,E2 -4876.432} C_VEL
LIN {X 0,Y 527.261,Z 409.276,A -85,B 0,C 180,E1 -4878.196,E2 -4878.196} C_VEL
LIN {X 0,Y 525.187,Z 397.562,A -85,B 0,C 180,E1 -4878.472,E2 -4878.472} C_VEL
LIN {X 0,Y 525.801,Z 375.209,A -85,B 0,C 180,E1 -4881.566,E2 -4881.566} C_VEL
LIN {X 0,Y 526.536,Z 353.264,A -85,B 0,C 180,E1 -4884.673,E2 -4884.673} C_VEL
LIN {X 0,Y 526.017,Z 349.055,A -85,B 0,C 180,E1 -4885.312,E2 -4885.312} C_VEL
LIN {X 0,Y 524.749,Z 343.526,A -85,B 0,C 180,E1 -4886.19,E2 -4886.19} C_VEL
LIN {X 0,Y 524.029,Z 341.796,A -85,B 0,C 180,E1 -4886.557,E2 -4886.557} C_VEL
LIN {X 0,Y 522.946,Z 340.817,A -85,B 0,C 180,E1 -4886.95,E2 -4886.95} C_VEL
LIN {X 0,Y 520.338,Z 340.296,A -85,B 0,C 180,E1 -4887.767,E2 -4887.767} C_VEL
LIN {X 0,Y 517.929,Z 340.596,A -85,B 0,C 180,E1 -4888.63,E2 -4888.63} C_VEL
LIN {X 0,Y 516.927,Z 340.723,A -85,B 0,C 180,E1 -4889.297,E2 -4889.297} C_VEL
LIN {X 0,Y 516.839,Z 340.73,A -85,B 0,C 180,E1 -4889.523,E2 -4889.523} C_VEL
LIN {X 0,Y 516.864,Z 340.727,A -85,B 0,C 180,E1 -4892.537,E2 -4892.537} C_VEL
LIN {X 0,Y 516.828,Z 340.729,A -85,B 0,C 180,E1 -4895.323,E2 -4895.323} C_VEL
LIN {X 0,Y 516.859,Z 340.725,A -85,B 0,C 180,E1 -4898.718,E2 -4898.718} C_VEL
LIN {X 0,Y 516.831,Z 340.731,A -85,B 0,C 180,E1 -4901.783,E2 -4901.783} C_VEL
LIN {X 0,Y 516.897,Z 340.72,A -85,B 0,C 180,E1 -4905.007,E2 -4905.007} C_VEL
LIN {X 0,Y 516.829,Z 340.732,A -85,B 0,C 180,E1 -4908.41,E2 -4908.41} C_VEL
LIN {X 0,Y 516.859,Z 340.723,A -85,B 0,C 180,E1 -4911.282,E2 -4911.282} C_VEL
LIN {X 0,Y 516.828,Z 340.73,A -85,B 0,C 180,E1 -4914.677,E2 -4914.677} C_VEL
LIN {X 0,Y 516.864,Z 340.728,A -85,B 0,C 180,E1 -4917.462,E2 -4917.462} C_VEL
LIN {X 0,Y 516.84,Z 340.719,A -85,B 0,C 180,E1 -4920.491,E2 -4920.491} C_VEL
LIN {X 0,Y 516.896,Z 340.981,A -85,B 0,C 180,E1 -4920.945,E2 -4920.945} C_VEL
LIN {X 0,Y 520.235,Z 355.076,A -85,B 0,C 180,E1 -4922.935,E2 -4922.935} C_VEL
LIN {X 0,Y 519.697,Z 376.671,A -85,B 0,C 180,E1 -4925.64,E2 -4925.64} C_VEL
LIN {X 0,Y 519.202,Z 398.257,A -85,B 0,C 180,E1 -4928.251,E2 -4928.251} C_VEL
LIN {X 0,Y 521.937,Z 413.106,A -85,B 0,C 180,E1 -4928.601,E2 -4928.601} C_VEL
LIN {X 0,Y 520.862,Z 564.936,A -85,B 0,C 180,E1 -4930.766,E2 -4930.766} C_VEL
LIN {X 0,Y 520.515,Z 580.486,A -85,B 0,C 180,E1 -4931.143,E2 -4931.143} C_VEL
LIN {X 0,Y 520.144,Z 594.664,A -85,B 0,C 180,E1 -4931.64,E2 -4931.64} C_VEL
LIN {X 0,Y 519.745,Z 608.714,A -85,B 0,C 180,E1 -4932.287,E2 -4932.287} C_VEL
LIN {X 0,Y 519.17,Z 622.418,A -85,B 0,C 180,E1 -4933.079,E2 -4933.079} C_VEL
LIN {X 0,Y 518.666,Z 635.138,A -85,B 0,C 180,E1 -4933.984,E2 -4933.984} C_VEL
LIN {X 0,Y 518.136,Z 647.738,A -85,B 0,C 180,E1 -4935.065,E2 -4935.065} C_VEL
LIN {X 0,Y 517.672,Z 659.293,A -85,B 0,C 180,E1 -4936.256,E2 -4936.256} C_VEL
LIN {X 0,Y 517.285,Z 669.029,A -85,B 0,C 180,E1 -4937.445,E2 -4937.445} C_VEL
LIN {X 0,Y 516.997,Z 678.559,A -85,B 0,C 180,E1 -4938.83,E2 -4938.83} C_VEL
LIN {X 0,Y 516.664,Z 686.49,A -85,B 0,C 180,E1 -4940.21,E2 -4940.21} C_VEL
LIN {X 0,Y 516.543,Z 692.197,A -85,B 0,C 180,E1 -4941.392,E2 -4941.392} C_VEL
LIN {X 0,Y 516.393,Z 698.397,A -85,B 0,C 180,E1 -4942.964,E2 -4942.964} C_VEL
LIN {X 0,Y 516.372,Z 703.269,A -85,B 0,C 180,E1 -4944.533,E2 -4944.533} C_VEL
LIN {X 0,Y 516.307,Z 706.826,A -85,B 0,C 180,E1 -4946.097,E2 -4946.097} C_VEL
LIN {X 0,Y 516.258,Z 709.128,A -85,B 0,C 180,E1 -4947.659,E2 -4947.659} C_VEL
LIN {X 0,Y 516.156,Z 710.268,A -85,B 0,C 180,E1 -4949.22,E2 -4949.22} C_VEL
LIN {X 0,Y 516.152,Z 710.493,A -85,B 0,C 180,E1 -4950,E2 -4950} C_VEL
LIN {X 0,Y 516.19,Z 709.94,A -85,B 0,C 180,E1 -4951.56,E2 -4951.56} C_VEL
LIN {X 0,Y 516.273,Z 708.224,A -85,B 0,C 180,E1 -4953.121,E2 -4953.121} C_VEL
LIN {X 0,Y 516.308,Z 706.99,A -85,B 0,C 180,E1 -4953.902,E2 -4953.902} C_VEL
LIN {X 0,Y 516.365,Z 702.413,A -85,B 0,C 180,E1 -4955.859,E2 -4955.859} C_VEL
LIN {X 0,Y 516.429,Z 697.32,A -85,B 0,C 180,E1 -4957.428,E2 -4957.428} C_VEL
LIN {X 0,Y 516.573,Z 690.819,A -85,B 0,C 180,E1 -4959.001,E2 -4959.001} C_VEL
LIN {X 0,Y 516.87,Z 682.663,A -85,B 0,C 180,E1 -4960.577,E2 -4960.577} C_VEL
LIN {X 0,Y 517.08,Z 674.547,A -85,B 0,C 180,E1 -4961.873,E2 -4961.873} C_VEL
LIN {X 0,Y 517.456,Z 665.081,A -85,B 0,C 180,E1 -4963.15,E2 -4963.15} C_VEL
LIN {X 0,Y 517.861,Z 654.637,A -85,B 0,C 180,E1 -4964.34,E2 -4964.34} C_VEL
LIN {X 0,Y 518.4,Z 643.104,A -85,B 0,C 180,E1 -4965.445,E2 -4965.445} C_VEL
LIN {X 0,Y 518.818,Z 631.079,A -85,B 0,C 180,E1 -4966.416,E2 -4966.416} C_VEL
LIN {X 0,Y 519.402,Z 617.448,A -85,B 0,C 180,E1 -4967.318,E2 -4967.318} C_VEL
LIN {X 0,Y 519.881,Z 603.504,A -85,B 0,C 180,E1 -4968.064,E2 -4968.064} C_VEL
LIN {X 0,Y 520.326,Z 588.514,A -85,B 0,C 180,E1 -4968.685,E2 -4968.685} C_VEL
LIN {X 0,Y 520.683,Z 573.396,A -85,B 0,C 180,E1 -4969.141,E2 -4969.141} C_VEL
LIN {X 0,Y 520.942,Z 557.137,A -85,B 0,C 180,E1 -4969.457,E2 -4969.457} C_VEL
LIN {X 0,Y 521.892,Z 412.51,A -85,B 0,C 180,E1 -4971.5,E2 -4971.5} C_VEL
LIN {X 0,Y 519.163,Z 398.231,A -85,B 0,C 180,E1 -4971.839,E2 -4971.839} C_VEL
LIN {X 0,Y 519.693,Z 375.675,A -85,B 0,C 180,E1 -4974.572,E2 -4974.572} C_VEL
LIN {X 0,Y 520.26,Z 356.03,A -85,B 0,C 180,E1 -4977.034,E2 -4977.034} C_VEL
LIN {X 0,Y 518.793,Z 348.756,A -85,B 0,C 180,E1 -4978.038,E2 -4978.038} C_VEL
LIN {X 0,Y 516.871,Z 340.897,A -85,B 0,C 180,E1 -4979.168,E2 -4979.168} C_VEL
LIN {X 0,Y 516.845,Z 340.732,A -85,B 0,C 180,E1 -4982.027,E2 -4982.027} C_VEL
LIN {X 0,Y 516.851,Z 340.727,A -85,B 0,C 180,E1 -4984.827,E2 -4984.827} C_VEL
LIN {X 0,Y 516.85,Z 340.733,A -85,B 0,C 180,E1 -4987.938,E2 -4987.938} C_VEL
LIN {X 0,Y 516.819,Z 340.729,A -85,B 0,C 180,E1 -4990.748,E2 -4990.748} C_VEL
LIN {X 0,Y 516.88,Z 340.729,A -85,B 0,C 180,E1 -4993.903,E2 -4993.903} C_VEL
LIN {X 0,Y 516.879,Z 340.727,A -85,B 0,C 180,E1 -4996.107,E2 -4996.107} C_VEL
LIN {X 0,Y 516.841,Z 340.729,A -85,B 0,C 180,E1 -4999.254,E2 -4999.254} C_VEL
LIN {X 0,Y 516.862,Z 340.729,A -85,B 0,C 180,E1 -5002.06,E2 -5002.06} C_VEL
LIN {X 0,Y 516.871,Z 340.721,A -85,B 0,C 180,E1 -5005.174,E2 -5005.174} C_VEL
LIN {X 0,Y 516.873,Z 340.723,A -85,B 0,C 180,E1 -5007.975,E2 -5007.975} C_VEL
LIN {X 0,Y 516.921,Z 340.716,A -85,B 0,C 180,E1 -5010.695,E2 -5010.695} C_VEL
LIN {X 0,Y 516.879,Z 340.727,A -85,B 0,C 180,E1 -5013.818,E2 -5013.818} C_VEL
LIN {X 0,Y 516.859,Z 340.722,A -85,B 0,C 180,E1 -5016.776,E2 -5016.776} C_VEL
LIN {X 0,Y 516.94,Z 340.721,A -85,B 0,C 180,E1 -5019.732,E2 -5019.732} C_VEL
LIN {X 0,Y 516.896,Z 340.714,A -85,B 0,C 180,E1 -5022.595,E2 -5022.595} C_VEL
LIN {X 0,Y 516.944,Z 340.713,A -85,B 0,C 180,E1 -5025.03,E2 -5025.03} C_VEL
LIN {X 0,Y 516.967,Z 340.705,A -85,B 0,C 180,E1 -5028.234,E2 -5028.234} C_VEL
LIN {X 0,Y 516.956,Z 340.717,A -85,B 0,C 180,E1 -5031.399,E2 -5031.399} C_VEL
LIN {X 0,Y 517.008,Z 340.705,A -85,B 0,C 180,E1 -5033.757,E2 -5033.757} C_VEL
LIN {X 0,Y 517.082,Z 340.701,A -85,B 0,C 180,E1 -5037.663,E2 -5037.663} C_VEL
LIN {X 0,Y 517.091,Z 340.692,A -85,B 0,C 180,E1 -5040.779,E2 -5040.779} C_VEL
LIN {X 0,Y 516.986,Z 340.708,A -85,B 0,C 180,E1 -5043.117,E2 -5043.117} C_VEL
LIN {X 0,Y 516.995,Z 340.704,A -85,B 0,C 180,E1 -5046.243,E2 -5046.243} C_VEL
LIN {X 0,Y 516.948,Z 340.717,A -85,B 0,C 180,E1 -5049.389,E2 -5049.389} C_VEL
LIN {X 0,Y 516.953,Z 340.711,A -85,B 0,C 180,E1 -5051.807,E2 -5051.807} C_VEL
LIN {X 0,Y 516.945,Z 340.714,A -85,B 0,C 180,E1 -5055.146,E2 -5055.146} C_VEL
LIN {X 0,Y 516.917,Z 340.714,A -85,B 0,C 180,E1 -5058.222,E2 -5058.222} C_VEL
LIN {X 0,Y 516.913,Z 340.714,A -85,B 0,C 180,E1 -5060.701,E2 -5060.701} C_VEL
LIN {X 0,Y 516.891,Z 340.716,A -85,B 0,C 180,E1 -5064.073,E2 -5064.073} C_VEL
LIN {X 0,Y 516.925,Z 340.716,A -85,B 0,C 180,E1 -5066.658,E2 -5066.658} C_VEL
LIN {X 0,Y 516.912,Z 340.716,A -85,B 0,C 180,E1 -5069.524,E2 -5069.524} C_VEL
LIN {X 0,Y 516.896,Z 340.721,A -85,B 0,C 180,E1 -5072.543,E2 -5072.543} C_VEL
LIN {X 0,Y 516.866,Z 340.728,A -85,B 0,C 180,E1 -5075.33,E2 -5075.33} C_VEL
LIN {X 0,Y 516.882,Z 340.718,A -85,B 0,C 180,E1 -5077.943,E2 -5077.943} C_VEL
LIN {X 0,Y 516.886,Z 340.708,A -85,B 0,C 180,E1 -5080.741,E2 -5080.741} C_VEL
LIN {X 0,Y 516.885,Z 340.723,A -85,B 0,C 180,E1 -5082.831,E2 -5082.831} C_VEL
LIN {X 0,Y 516.923,Z 340.717,A -85,B 0,C 180,E1 -5085.01,E2 -5085.01} C_VEL
LIN {X 0,Y 516.917,Z 340.715,A -85,B 0,C 180,E1 -5088.398,E2 -5088.398} C_VEL
LIN {X 0,Y 516.884,Z 340.726,A -85,B 0,C 180,E1 -5091.284,E2 -5091.284} C_VEL
LIN {X 0,Y 516.871,Z 340.724,A -85,B 0,C 180,E1 -5094.22,E2 -5094.22} C_VEL
LIN {X 0,Y 516.895,Z 340.727,A -85,B 0,C 180,E1 -5097.053,E2 -5097.053} C_VEL
LIN {X 0,Y 516.893,Z 340.725,A -85,B 0,C 180,E1 -5099.796,E2 -5099.796} C_VEL
LIN {X 0,Y 516.94,Z 340.906,A -85,B 0,C 180,E1 -5101.323,E2 -5101.323} C_VEL
LIN {X 0,Y 520.864,Z 356.1,A -85,B 0,C 180,E1 -5103.43,E2 -5103.43} C_VEL
LIN {X 0,Y 520.008,Z 378.702,A -85,B 0,C 180,E1 -5106.08,E2 -5106.08} C_VEL
LIN {X 0,Y 519.404,Z 397.52,A -85,B 0,C 180,E1 -5108.244,E2 -5108.244} C_VEL
LIN {X 0,Y 519.638,Z 399.766,A -85,B 0,C 180,E1 -5108.342,E2 -5108.342} C_VEL
LIN {X 0,Y 521.742,Z 412.691,A -85,B 0,C 180,E1 -5108.621,E2 -5108.621} C_VEL
LIN {X 0,Y 520.499,Z 564.295,A -85,B 0,C 180,E1 -5110.825,E2 -5110.825} C_VEL
LIN {X 0,Y 520.22,Z 580.074,A -85,B 0,C 180,E1 -5111.209,E2 -5111.209} C_VEL
LIN {X 0,Y 519.852,Z 594.92,A -85,B 0,C 180,E1 -5111.731,E2 -5111.731} C_VEL
LIN {X 0,Y 519.41,Z 608.887,A -85,B 0,C 180,E1 -5112.377,E2 -5112.377} C_VEL
LIN {X 0,Y 518.926,Z 622.572,A -85,B 0,C 180,E1 -5113.173,E2 -5113.173} C_VEL
LIN {X 0,Y 518.489,Z 635.163,A -85,B 0,C 180,E1 -5114.069,E2 -5114.069} C_VEL
LIN {X 0,Y 518.039,Z 646.858,A -85,B 0,C 180,E1 -5115.063,E2 -5115.063} C_VEL
LIN {X 0,Y 517.584,Z 658.63,A -85,B 0,C 180,E1 -5116.254,E2 -5116.254} C_VEL
LIN {X 0,Y 517.213,Z 668.517,A -85,B 0,C 180,E1 -5117.443,E2 -5117.443} C_VEL
LIN {X 0,Y 516.923,Z 678.2,A -85,B 0,C 180,E1 -5118.829,E2 -5118.829} C_VEL
LIN {X 0,Y 516.626,Z 686.247,A -85,B 0,C 180,E1 -5120.21,E2 -5120.21} C_VEL
LIN {X 0,Y 516.479,Z 693.75,A -85,B 0,C 180,E1 -5121.786,E2 -5121.786} C_VEL
LIN {X 0,Y 516.391,Z 698.348,A -85,B 0,C 180,E1 -5122.964,E2 -5122.964} C_VEL
LIN {X 0,Y 516.352,Z 703.217,A -85,B 0,C 180,E1 -5124.533,E2 -5124.533} C_VEL
LIN {X 0,Y 516.293,Z 706.777,A -85,B 0,C 180,E1 -5126.097,E2 -5126.097} C_VEL
LIN {X 0,Y 516.258,Z 709.117,A -85,B 0,C 180,E1 -5127.659,E2 -5127.659} C_VEL
LIN {X 0,Y 516.156,Z 710.289,A -85,B 0,C 180,E1 -5129.22,E2 -5129.22} C_VEL
LIN {X 0,Y 516.156,Z 710.288,A -85,B 0,C 180,E1 -5130.78,E2 -5130.78} C_VEL
LIN {X 0,Y 516.258,Z 709.111,A -85,B 0,C 180,E1 -5132.341,E2 -5132.341} C_VEL
LIN {X 0,Y 516.293,Z 706.768,A -85,B 0,C 180,E1 -5133.903,E2 -5133.903} C_VEL
LIN {X 0,Y 516.352,Z 703.205,A -85,B 0,C 180,E1 -5135.467,E2 -5135.467} C_VEL
LIN {X 0,Y 516.391,Z 698.325,A -85,B 0,C 180,E1 -5137.036,E2 -5137.036} C_VEL
LIN {X 0,Y 516.541,Z 691.991,A -85,B 0,C 180,E1 -5138.608,E2 -5138.608} C_VEL
LIN {X 0,Y 516.728,Z 684.015,A -85,B 0,C 180,E1 -5140.184,E2 -5140.184} C_VEL
LIN {X 0,Y 516.96,Z 675.498,A -85,B 0,C 180,E1 -5141.568,E2 -5141.568} C_VEL
LIN {X 0,Y 517.328,Z 665.21,A -85,B 0,C 180,E1 -5142.953,E2 -5142.953} C_VEL
LIN {X 0,Y 517.671,Z 654.669,A -85,B 0,C 180,E1 -5144.145,E2 -5144.145} C_VEL
LIN {X 0,Y 518.117,Z 642.435,A -85,B 0,C 180,E1 -5145.3,E2 -5145.3} C_VEL
LIN {X 0,Y 518.602,Z 629.231,A -85,B 0,C 180,E1 -5146.332,E2 -5146.332} C_VEL
LIN {X 0,Y 519.066,Z 616.945,A -85,B 0,C 180,E1 -5147.127,E2 -5147.127} C_VEL
LIN {X 0,Y 519.489,Z 602.746,A -85,B 0,C 180,E1 -5147.875,E2 -5147.875} C_VEL
LIN {X 0,Y 519.912,Z 587.103,A -85,B 0,C 180,E1 -5148.508,E2 -5148.508} C_VEL
LIN {X 0,Y 520.259,Z 571.614,A -85,B 0,C 180,E1 -5148.959,E2 -5148.959} C_VEL
LIN {X 0,Y 520.454,Z 555.807,A -85,B 0,C 180,E1 -5149.256,E2 -5149.256} C_VEL
LIN {X 0,Y 521.501,Z 418.471,A -85,B 0,C 180,E1 -5151.241,E2 -5151.241} C_VEL
LIN {X 0,Y 521.42,Z 410.782,A -85,B 0,C 180,E1 -5151.363,E2 -5151.363} C_VEL
LIN {X 0,Y 519.29,Z 397.895,A -85,B 0,C 180,E1 -5151.668,E2 -5151.668} C_VEL
LIN {X 0,Y 520.227,Z 371.103,A -85,B 0,C 180,E1 -5154.759,E2 -5154.759} C_VEL
LIN {X 0,Y 520.84,Z 357.011,A -85,B 0,C 180,E1 -5156.442,E2 -5156.442} C_VEL
LIN {X 0,Y 519.084,Z 348.843,A -85,B 0,C 180,E1 -5157.567,E2 -5157.567} C_VEL
LIN {X 0,Y 516.925,Z 340.86,A -85,B 0,C 180,E1 -5158.775,E2 -5158.775} C_VEL
LIN {X 0,Y 516.89,Z 340.728,A -85,B 0,C 180,E1 -5161.11,E2 -5161.11} C_VEL
LIN {X 0,Y 516.912,Z 340.719,A -85,B 0,C 180,E1 -5163.967,E2 -5163.967} C_VEL
LIN {X 0,Y 516.879,Z 340.729,A -85,B 0,C 180,E1 -5166.746,E2 -5166.746} C_VEL
LIN {X 0,Y 516.883,Z 340.723,A -85,B 0,C 180,E1 -5169.721,E2 -5169.721} C_VEL
LIN {X 0,Y 516.912,Z 340.719,A -85,B 0,C 180,E1 -5171.775,E2 -5171.775} C_VEL
LIN {X 0,Y 516.896,Z 340.725,A -85,B 0,C 180,E1 -5175.007,E2 -5175.007} C_VEL
LIN {X 0,Y 516.911,Z 340.724,A -85,B 0,C 180,E1 -5178.399,E2 -5178.399} C_VEL
LIN {X 0,Y 516.879,Z 340.724,A -85,B 0,C 180,E1 -5181.284,E2 -5181.284} C_VEL
LIN {X 0,Y 516.867,Z 340.73,A -85,B 0,C 180,E1 -5184.219,E2 -5184.219} C_VEL
LIN {X 0,Y 516.888,Z 340.724,A -85,B 0,C 180,E1 -5187.053,E2 -5187.053} C_VEL
LIN {X 0,Y 516.866,Z 340.73,A -85,B 0,C 180,E1 -5189.795,E2 -5189.795} C_VEL
LIN {X 0,Y 516.877,Z 340.872,A -85,B 0,C 180,E1 -5192.766,E2 -5192.766} C_VEL
LIN {X 0,Y 519.351,Z 351.031,A -85,B 0,C 180,E1 -5194.524,E2 -5194.524} C_VEL
LIN {X 0,Y 519.985,Z 355.43,A -85,B 0,C 180,E1 -5195.229,E2 -5195.229} C_VEL
LIN {X 0,Y 518.981,Z 379.652,A -85,B 0,C 180,E1 -5198.748,E2 -5198.748} C_VEL
LIN {X 0,Y 518.439,Z 397.779,A -85,B 0,C 180,E1 -5201.296,E2 -5201.296} C_VEL
LIN {X 0,Y 520.684,Z 410.59,A -85,B 0,C 180,E1 -5201.613,E2 -5201.613} C_VEL
LIN {X 0,Y 519.502,Z 537.731,A -85,B 0,C 180,E1 -5203.558,E2 -5203.558} C_VEL
LIN {X 0,Y 519.218,Z 552.076,A -85,B 0,C 180,E1 -5203.935,E2 -5203.935} C_VEL
LIN {X 0,Y 518.96,Z 566.451,A -85,B 0,C 180,E1 -5204.487,E2 -5204.487} C_VEL
LIN {X 0,Y 518.592,Z 580.025,A -85,B 0,C 180,E1 -5205.179,E2 -5205.179} C_VEL
LIN {X 0,Y 518.174,Z 592.263,A -85,B 0,C 180,E1 -5205.97,E2 -5205.97} C_VEL
LIN {X 0,Y 517.782,Z 604.58,A -85,B 0,C 180,E1 -5206.959,E2 -5206.959} C_VEL
LIN {X 0,Y 517.43,Z 614.653,A -85,B 0,C 180,E1 -5207.944,E2 -5207.944} C_VEL
LIN {X 0,Y 517.139,Z 623.969,A -85,B 0,C 180,E1 -5209.032,E2 -5209.032} C_VEL
LIN {X 0,Y 516.874,Z 632.405,A -85,B 0,C 180,E1 -5210.214,E2 -5210.214} C_VEL
LIN {X 0,Y 516.637,Z 640.437,A -85,B 0,C 180,E1 -5211.591,E2 -5211.591} C_VEL
LIN {X 0,Y 516.469,Z 646.902,A -85,B 0,C 180,E1 -5212.965,E2 -5212.965} C_VEL
LIN {X 0,Y 516.438,Z 651.318,A -85,B 0,C 180,E1 -5214.142,E2 -5214.142} C_VEL
LIN {X 0,Y 516.276,Z 654.833,A -85,B 0,C 180,E1 -5215.315,E2 -5215.315} C_VEL
LIN {X 0,Y 516.343,Z 656.73,A -85,B 0,C 180,E1 -5216.098,E2 -5216.098} C_VEL
LIN {X 0,Y 516.26,Z 659.416,A -85,B 0,C 180,E1 -5217.659,E2 -5217.659} C_VEL
LIN {X 0,Y 516.156,Z 660.777,A -85,B 0,C 180,E1 -5219.22,E2 -5219.22} C_VEL
LIN {X 0,Y 516.157,Z 660.794,A -85,B 0,C 180,E1 -5220.78,E2 -5220.78} C_VEL
LIN {X 0,Y 516.259,Z 659.51,A -85,B 0,C 180,E1 -5222.341,E2 -5222.341} C_VEL
LIN {X 0,Y 516.343,Z 656.872,A -85,B 0,C 180,E1 -5223.902,E2 -5223.902} C_VEL
LIN {X 0,Y 516.387,Z 652.797,A -85,B 0,C 180,E1 -5225.467,E2 -5225.467} C_VEL
LIN {X 0,Y 516.419,Z 648.775,A -85,B 0,C 180,E1 -5226.631,E2 -5226.631} C_VEL
LIN {X 0,Y 516.533,Z 643.718,A -85,B 0,C 180,E1 -5227.82,E2 -5227.82} C_VEL
LIN {X 0,Y 516.755,Z 636.487,A -85,B 0,C 180,E1 -5229.196,E2 -5229.196} C_VEL
LIN {X 0,Y 517.007,Z 627.514,A -85,B 0,C 180,E1 -5230.575,E2 -5230.575} C_VEL
LIN {X 0,Y 517.322,Z 618.051,A -85,B 0,C 180,E1 -5231.758,E2 -5231.758} C_VEL
LIN {X 0,Y 517.662,Z 607.626,A -85,B 0,C 180,E1 -5232.845,E2 -5232.845} C_VEL
LIN {X 0,Y 518.057,Z 596.006,A -85,B 0,C 180,E1 -5233.834,E2 -5233.834} C_VEL
LIN {X 0,Y 518.449,Z 584.779,A -85,B 0,C 180,E1 -5234.624,E2 -5234.624} C_VEL
LIN {X 0,Y 518.801,Z 572.603,A -85,B 0,C 180,E1 -5235.317,E2 -5235.317} C_VEL
LIN {X 0,Y 519.17,Z 558.615,A -85,B 0,C 180,E1 -5235.934,E2 -5235.934} C_VEL
LIN {X 0,Y 519.45,Z 543.939,A -85,B 0,C 180,E1 -5236.403,E2 -5236.403} C_VEL
LIN {X 0,Y 519.661,Z 528.917,A -85,B 0,C 180,E1 -5236.702,E2 -5236.702} C_VEL
LIN {X 0,Y 520.453,Z 409.425,A -85,B 0,C 180,E1 -5238.452,E2 -5238.452} C_VEL
LIN {X 0,Y 518.284,Z 397.688,A -85,B 0,C 180,E1 -5238.733,E2 -5238.733} C_VEL
LIN {X 0,Y 518.887,Z 378.183,A -85,B 0,C 180,E1 -5241.451,E2 -5241.451} C_VEL
LIN {X 0,Y 519.648,Z 356.369,A -85,B 0,C 180,E1 -5244.575,E2 -5244.575} C_VEL
LIN {X 0,Y 519.67,Z 353.274,A -85,B 0,C 180,E1 -5245.027,E2 -5245.027} C_VEL
LIN {X 0,Y 516.934,Z 341.182,A -85,B 0,C 180,E1 -5246.985,E2 -5246.985} C_VEL
LIN {X 0,Y 516.874,Z 340.728,A -85,B 0,C 180,E1 -5247.207,E2 -5247.207} C_VEL
LIN {X 0,Y 516.839,Z 340.73,A -85,B 0,C 180,E1 -5249.523,E2 -5249.523} C_VEL
LIN {X 0,Y 516.159,Z 340.818,A -85,B 0,C 180,E1 -5250.173,E2 -5250.173} C_VEL
LIN {X 0,Y 513.318,Z 341.168,A -85,B 0,C 180,E1 -5251.229,E2 -5251.229} C_VEL
LIN {X 0,Y 510.926,Z 341.471,A -85,B 0,C 180,E1 -5252.08,E2 -5252.08} C_VEL
LIN {X 0,Y 509.899,Z 341.594,A -85,B 0,C 180,E1 -5252.737,E2 -5252.737} C_VEL
LIN {X 0,Y 509.815,Z 341.603,A -85,B 0,C 180,E1 -5252.959,E2 -5252.959} C_VEL
LIN {X 0,Y 509.779,Z 341.609,A -85,B 0,C 180,E1 -5255.571,E2 -5255.571} C_VEL
LIN {X 0,Y 509.808,Z 341.607,A -85,B 0,C 180,E1 -5258.342,E2 -5258.342} C_VEL
LIN {X 0,Y 509.783,Z 341.606,A -85,B 0,C 180,E1 -5261.433,E2 -5261.433} C_VEL
LIN {X 0,Y 509.835,Z 341.601,A -85,B 0,C 180,E1 -5264.67,E2 -5264.67} C_VEL
LIN {X 0,Y 509.783,Z 341.601,A -85,B 0,C 180,E1 -5267.505,E2 -5267.505} C_VEL
LIN {X 0,Y 509.81,Z 341.603,A -85,B 0,C 180,E1 -5270.644,E2 -5270.644} C_VEL
LIN {X 0,Y 509.761,Z 341.608,A -85,B 0,C 180,E1 -5273.641,E2 -5273.641} C_VEL
LIN {X 0,Y 509.825,Z 341.606,A -85,B 0,C 180,E1 -5276.536,E2 -5276.536} C_VEL
LIN {X 0,Y 509.802,Z 341.602,A -85,B 0,C 180,E1 -5279.331,E2 -5279.331} C_VEL
LIN {X 0,Y 509.809,Z 341.771,A -85,B 0,C 180,E1 -5280.648,E2 -5280.648} C_VEL
LIN {X 0,Y 513.453,Z 356.969,A -85,B 0,C 180,E1 -5282.836,E2 -5282.836} C_VEL
LIN {X 0,Y 512.8,Z 379.8,A -85,B 0,C 180,E1 -5285.722,E2 -5285.722} C_VEL
LIN {X 0,Y 512.364,Z 398.06,A -85,B 0,C 180,E1 -5287.941,E2 -5287.941} C_VEL
LIN {X 0,Y 515.313,Z 413.76,A -85,B 0,C 180,E1 -5288.323,E2 -5288.323} C_VEL
LIN {X 0,Y 514.181,Z 564.499,A -85,B 0,C 180,E1 -5290.5,E2 -5290.5} C_VEL
LIN {X 0,Y 513.817,Z 579.563,A -85,B 0,C 180,E1 -5290.862,E2 -5290.862} C_VEL
LIN {X 0,Y 513.372,Z 594.612,A -85,B 0,C 180,E1 -5291.389,E2 -5291.389} C_VEL
LIN {X 0,Y 512.948,Z 608.673,A -85,B 0,C 180,E1 -5292.044,E2 -5292.044} C_VEL
LIN {X 0,Y 512.355,Z 622.385,A -85,B 0,C 180,E1 -5292.847,E2 -5292.847} C_VEL
LIN {X 0,Y 511.797,Z 635.112,A -85,B 0,C 180,E1 -5293.763,E2 -5293.763} C_VEL
LIN {X 0,Y 511.226,Z 647.717,A -85,B 0,C 180,E1 -5294.859,E2 -5294.859} C_VEL
LIN {X 0,Y 510.723,Z 659.275,A -85,B 0,C 180,E1 -5296.065,E2 -5296.065} C_VEL
LIN {X 0,Y 510.279,Z 669.012,A -85,B 0,C 180,E1 -5297.269,E2 -5297.269} C_VEL
LIN {X 0,Y 509.971,Z 678.662,A -85,B 0,C 180,E1 -5298.694,E2 -5298.694} C_VEL
LIN {X 0,Y 509.637,Z 686.488,A -85,B 0,C 180,E1 -5300.074,E2 -5300.074} C_VEL
LIN {X 0,Y 509.433,Z 693.89,A -85,B 0,C 180,E1 -5301.671,E2 -5301.671} C_VEL
LIN {X 0,Y 509.257,Z 699.89,A -85,B 0,C 180,E1 -5303.303,E2 -5303.303} C_VEL
LIN {X 0,Y 509.281,Z 703.24,A -85,B 0,C 180,E1 -5304.457,E2 -5304.457} C_VEL
LIN {X 0,Y 509.2,Z 706.79,A -85,B 0,C 180,E1 -5306.043,E2 -5306.043} C_VEL
LIN {X 0,Y 509.158,Z 709.126,A -85,B 0,C 180,E1 -5307.627,E2 -5307.627} C_VEL
LIN {X 0,Y 509.07,Z 710.307,A -85,B 0,C 180,E1 -5309.209,E2 -5309.209} C_VEL
LIN {X 0,Y 509.071,Z 710.333,A -85,B 0,C 180,E1 -5310.791,E2 -5310.791} C_VEL
LIN {X 0,Y 509.159,Z 709.213,A -85,B 0,C 180,E1 -5312.373,E2 -5312.373} C_VEL
LIN {X 0,Y 509.201,Z 706.949,A -85,B 0,C 180,E1 -5313.957,E2 -5313.957} C_VEL
LIN {X 0,Y 509.279,Z 703.48,A -85,B 0,C 180,E1 -5315.543,E2 -5315.543} C_VEL
LIN {X 0,Y 509.319,Z 698.732,A -85,B 0,C 180,E1 -5317.134,E2 -5317.134} C_VEL
LIN {X 0,Y 509.471,Z 692.573,A -85,B 0,C 180,E1 -5318.728,E2 -5318.728} C_VEL
LIN {X 0,Y 509.738,Z 684.833,A -85,B 0,C 180,E1 -5320.325,E2 -5320.325} C_VEL
LIN {X 0,Y 509.988,Z 676.339,A -85,B 0,C 180,E1 -5321.765,E2 -5321.765} C_VEL
LIN {X 0,Y 510.402,Z 666.651,A -85,B 0,C 180,E1 -5323.132,E2 -5323.132} C_VEL
LIN {X 0,Y 510.879,Z 656.515,A -85,B 0,C 180,E1 -5324.337,E2 -5324.337} C_VEL
LIN {X 0,Y 511.424,Z 645.146,A -85,B 0,C 180,E1 -5325.475,E2 -5325.475} C_VEL
LIN {X 0,Y 511.931,Z 632.281,A -85,B 0,C 180,E1 -5326.551,E2 -5326.551} C_VEL
LIN {X 0,Y 512.555,Z 619.095,A -85,B 0,C 180,E1 -5327.454,E2 -5327.454} C_VEL
LIN {X 0,Y 513.071,Z 604.512,A -85,B 0,C 180,E1 -5328.261,E2 -5328.261} C_VEL
LIN {X 0,Y 513.559,Z 589.483,A -85,B 0,C 180,E1 -5328.902,E2 -5328.902} C_VEL
LIN {X 0,Y 513.981,Z 574.189,A -85,B 0,C 180,E1 -5329.377,E2 -5329.377} C_VEL
LIN {X 0,Y 514.251,Z 558.75,A -85,B 0,C 180,E1 -5329.692,E2 -5329.692} C_VEL
LIN {X 0,Y 515.26,Z 413.478,A -85,B 0,C 180,E1 -5331.774,E2 -5331.774} C_VEL
LIN {X 0,Y 512.325,Z 398.209,A -85,B 0,C 180,E1 -5332.141,E2 -5332.141} C_VEL
LIN {X 0,Y 512.76,Z 380.532,A -85,B 0,C 180,E1 -5334.279,E2 -5334.279} C_VEL
LIN {X 0,Y 513.462,Z 357.678,A -85,B 0,C 180,E1 -5337.166,E2 -5337.166} C_VEL
LIN {X 0,Y 510.948,Z 346.23,A -85,B 0,C 180,E1 -5338.778,E2 -5338.778} C_VEL
LIN {X 0,Y 509.808,Z 341.738,A -85,B 0,C 180,E1 -5339.454,E2 -5339.454} C_VEL
LIN {X 0,Y 509.831,Z 341.603,A -85,B 0,C 180,E1 -5342.521,E2 -5342.521} C_VEL
LIN {X 0,Y 509.788,Z 341.609,A -85,B 0,C 180,E1 -5345.381,E2 -5345.381} C_VEL
LIN {X 0,Y 509.807,Z 341.604,A -85,B 0,C 180,E1 -5348.342,E2 -5348.342} C_VEL
LIN {X 0,Y 509.782,Z 341.608,A -85,B 0,C 180,E1 -5351.433,E2 -5351.433} C_VEL
LIN {X 0,Y 509.839,Z 341.597,A -85,B 0,C 180,E1 -5354.67,E2 -5354.67} C_VEL
LIN {X 0,Y 509.786,Z 341.61,A -85,B 0,C 180,E1 -5357.505,E2 -5357.505} C_VEL
LIN {X 0,Y 509.828,Z 341.598,A -85,B 0,C 180,E1 -5360.646,E2 -5360.646} C_VEL
LIN {X 0,Y 509.797,Z 341.61,A -85,B 0,C 180,E1 -5363.644,E2 -5363.644} C_VEL
LIN {X 0,Y 509.839,Z 341.598,A -85,B 0,C 180,E1 -5366.538,E2 -5366.538} C_VEL
LIN {X 0,Y 509.843,Z 341.597,A -85,B 0,C 180,E1 -5369.334,E2 -5369.334} C_VEL
LIN {X 0,Y 509.839,Z 341.597,A -85,B 0,C 180,E1 -5372.051,E2 -5372.051} C_VEL
LIN {X 0,Y 509.801,Z 341.602,A -85,B 0,C 180,E1 -5374.7,E2 -5374.7} C_VEL
LIN {X 0,Y 509.827,Z 341.602,A -85,B 0,C 180,E1 -5377.458,E2 -5377.458} C_VEL
LIN {X 0,Y 509.917,Z 341.594,A -85,B 0,C 180,E1 -5379.845,E2 -5379.845} C_VEL
LIN {X 0,Y 509.865,Z 341.593,A -85,B 0,C 180,E1 -5383.174,E2 -5383.174} C_VEL
LIN {X 0,Y 509.862,Z 341.603,A -85,B 0,C 180,E1 -5385.634,E2 -5385.634} C_VEL
LIN {X 0,Y 509.912,Z 341.584,A -85,B 0,C 180,E1 -5388.874,E2 -5388.874} C_VEL
LIN {X 0,Y 509.921,Z 341.589,A -85,B 0,C 180,E1 -5392.078,E2 -5392.078} C_VEL
LIN {X 0,Y 509.978,Z 341.575,A -85,B 0,C 180,E1 -5394.464,E2 -5394.464} C_VEL
LIN {X 0,Y 510.051,Z 341.578,A -85,B 0,C 180,E1 -5397.631,E2 -5397.631} C_VEL
LIN {X 0,Y 510.057,Z 341.568,A -85,B 0,C 180,E1 -5400,E2 -5400} C_VEL
LIN {X 0,Y 510.052,Z 341.566,A -85,B 0,C 180,E1 -5402.369,E2 -5402.369} C_VEL
LIN {X 0,Y 509.976,Z 341.584,A -85,B 0,C 180,E1 -5405.536,E2 -5405.536} C_VEL
LIN {X 0,Y 509.907,Z 341.584,A -85,B 0,C 180,E1 -5408.72,E2 -5408.72} C_VEL
LIN {X 0,Y 509.905,Z 341.588,A -85,B 0,C 180,E1 -5411.932,E2 -5411.932} C_VEL
LIN {X 0,Y 509.895,Z 341.593,A -85,B 0,C 180,E1 -5415.242,E2 -5415.242} C_VEL
LIN {X 0,Y 509.862,Z 341.593,A -85,B 0,C 180,E1 -5418.484,E2 -5418.484} C_VEL
LIN {X 0,Y 509.851,Z 341.597,A -85,B 0,C 180,E1 -5421.002,E2 -5421.002} C_VEL
LIN {X 0,Y 509.856,Z 341.593,A -85,B 0,C 180,E1 -5424.427,E2 -5424.427} C_VEL
LIN {X 0,Y 509.884,Z 341.598,A -85,B 0,C 180,E1 -5427.056,E2 -5427.056} C_VEL
LIN {X 0,Y 509.858,Z 341.592,A -85,B 0,C 180,E1 -5429.751,E2 -5429.751} C_VEL
LIN {X 0,Y 509.873,Z 341.598,A -85,B 0,C 180,E1 -5432.774,E2 -5432.774} C_VEL
LIN {X 0,Y 509.826,Z 341.602,A -85,B 0,C 180,E1 -5435.578,E2 -5435.578} C_VEL
LIN {X 0,Y 509.851,Z 341.594,A -85,B 0,C 180,E1 -5438.338,E2 -5438.338} C_VEL
LIN {X 0,Y 509.859,Z 341.594,A -85,B 0,C 180,E1 -5441.425,E2 -5441.425} C_VEL
LIN {X 0,Y 509.857,Z 341.601,A -85,B 0,C 180,E1 -5444.668,E2 -5444.668} C_VEL
LIN {X 0,Y 509.859,Z 341.592,A -85,B 0,C 180,E1 -5448.103,E2 -5448.103} C_VEL
LIN {X 0,Y 509.848,Z 341.602,A -85,B 0,C 180,E1 -5450.648,E2 -5450.648} C_VEL
LIN {X 0,Y 509.825,Z 341.602,A -85,B 0,C 180,E1 -5453.647,E2 -5453.647} C_VEL
LIN {X 0,Y 509.859,Z 341.601,A -85,B 0,C 180,E1 -5456.539,E2 -5456.539} C_VEL
LIN {X 0,Y 509.846,Z 341.603,A -85,B 0,C 180,E1 -5459.334,E2 -5459.334} C_VEL
LIN {X 0,Y 509.919,Z 341.813,A -85,B 0,C 180,E1 -5461.017,E2 -5461.017} C_VEL
LIN {X 0,Y 513.888,Z 357.079,A -85,B 0,C 180,E1 -5463.172,E2 -5463.172} C_VEL
LIN {X 0,Y 514.053,Z 360.673,A -85,B 0,C 180,E1 -5463.619,E2 -5463.619} C_VEL
LIN {X 0,Y 512.881,Z 388.537,A -85,B 0,C 180,E1 -5466.919,E2 -5466.919} C_VEL
LIN {X 0,Y 512.597,Z 397.497,A -85,B 0,C 180,E1 -5467.956,E2 -5467.956} C_VEL
LIN {X 0,Y 512.875,Z 399.947,A -85,B 0,C 180,E1 -5468.063,E2 -5468.063} C_VEL
LIN {X 0,Y 515.064,Z 413.558,A -85,B 0,C 180,E1 -5468.368,E2 -5468.368} C_VEL
LIN {X 0,Y 513.696,Z 565.435,A -85,B 0,C 180,E1 -5470.624,E2 -5470.624} C_VEL
LIN {X 0,Y 513.384,Z 580.815,A -85,B 0,C 180,E1 -5471.017,E2 -5471.017} C_VEL
LIN {X 0,Y 512.985,Z 595.239,A -85,B 0,C 180,E1 -5471.538,E2 -5471.538} C_VEL
LIN {X 0,Y 512.48,Z 609.883,A -85,B 0,C 180,E1 -5472.234,E2 -5472.234} C_VEL
LIN {X 0,Y 511.977,Z 623.349,A -85,B 0,C 180,E1 -5473.04,E2 -5473.04} C_VEL
LIN {X 0,Y 511.431,Z 637.031,A -85,B 0,C 180,E1 -5474.048,E2 -5474.048} C_VEL
LIN {X 0,Y 510.926,Z 649.449,A -85,B 0,C 180,E1 -5475.156,E2 -5475.156} C_VEL
LIN {X 0,Y 510.466,Z 661.596,A -85,B 0,C 180,E1 -5476.464,E2 -5476.464} C_VEL
LIN {X 0,Y 510.094,Z 671.026,A -85,B 0,C 180,E1 -5477.669,E2 -5477.669} C_VEL
LIN {X 0,Y 509.794,Z 680.241,A -85,B 0,C 180,E1 -5479.073,E2 -5479.073} C_VEL
LIN {X 0,Y 509.51,Z 687.871,A -85,B 0,C 180,E1 -5480.472,E2 -5480.472} C_VEL
LIN {X 0,Y 509.378,Z 694.992,A -85,B 0,C 180,E1 -5482.07,E2 -5482.07} C_VEL
LIN {X 0,Y 509.265,Z 700.581,A -85,B 0,C 180,E1 -5483.662,E2 -5483.662} C_VEL
LIN {X 0,Y 509.158,Z 704.797,A -85,B 0,C 180,E1 -5485.249,E2 -5485.249} C_VEL
LIN {X 0,Y 509.187,Z 707.755,A -85,B 0,C 180,E1 -5486.835,E2 -5486.835} C_VEL
LIN {X 0,Y 509.11,Z 709.511,A -85,B 0,C 180,E1 -5488.418,E2 -5488.418} C_VEL
LIN {X 0,Y 509.062,Z 710.107,A -85,B 0,C 180,E1 -5490,E2 -5490} C_VEL
LIN {X 0,Y 509.11,Z 709.498,A -85,B 0,C 180,E1 -5491.582,E2 -5491.582} C_VEL
LIN {X 0,Y 509.187,Z 707.729,A -85,B 0,C 180,E1 -5493.165,E2 -5493.165} C_VEL
LIN {X 0,Y 509.158,Z 704.76,A -85,B 0,C 180,E1 -5494.751,E2 -5494.751} C_VEL
LIN {X 0,Y 509.237,Z 700.524,A -85,B 0,C 180,E1 -5496.339,E2 -5496.339} C_VEL
LIN {X 0,Y 509.378,Z 694.9,A -85,B 0,C 180,E1 -5497.931,E2 -5497.931} C_VEL
LIN {X 0,Y 509.508,Z 687.721,A -85,B 0,C 180,E1 -5499.528,E2 -5499.528} C_VEL
LIN {X 0,Y 509.785,Z 680.03,A -85,B 0,C 180,E1 -5500.927,E2 -5500.927} C_VEL
LIN {X 0,Y 510.092,Z 670.732,A -85,B 0,C 180,E1 -5502.331,E2 -5502.331} C_VEL
LIN {X 0,Y 510.483,Z 659.454,A -85,B 0,C 180,E1 -5503.738,E2 -5503.738} C_VEL
LIN {X 0,Y 510.921,Z 647.82,A -85,B 0,C 180,E1 -5504.947,E2 -5504.947} C_VEL
LIN {X 0,Y 511.46,Z 634.98,A -85,B 0,C 180,E1 -5506.054,E2 -5506.054} C_VEL
LIN {X 0,Y 511.894,Z 622.29,A -85,B 0,C 180,E1 -5506.963,E2 -5506.963} C_VEL
LIN {X 0,Y 512.402,Z 608.483,A -85,B 0,C 180,E1 -5507.769,E2 -5507.769} C_VEL
LIN {X 0,Y 512.864,Z 594.56,A -85,B 0,C 180,E1 -5508.417,E2 -5508.417} C_VEL
LIN {X 0,Y 513.232,Z 579.249,A -85,B 0,C 180,E1 -5508.956,E2 -5508.956} C_VEL
LIN {X 0,Y 513.55,Z 563.793,A -85,B 0,C 180,E1 -5509.33,E2 -5509.33} C_VEL
LIN {X 0,Y 514.817,Z 412.368,A -85,B 0,C 180,E1 -5511.592,E2 -5511.592} C_VEL
LIN {X 0,Y 512.452,Z 398.011,A -85,B 0,C 180,E1 -5511.942,E2 -5511.942} C_VEL
LIN {X 0,Y 513.45,Z 372.863,A -85,B 0,C 180,E1 -5514.892,E2 -5514.892} C_VEL
LIN {X 0,Y 514.133,Z 358.883,A -85,B 0,C 180,E1 -5516.595,E2 -5516.595} C_VEL
LIN {X 0,Y 511.949,Z 349.25,A -85,B 0,C 180,E1 -5517.971,E2 -5517.971} C_VEL
LIN {X 0,Y 509.907,Z 341.726,A -85,B 0,C 180,E1 -5519.153,E2 -5519.153} C_VEL
LIN {X 0,Y 509.862,Z 341.602,A -85,B 0,C 180,E1 -5522.519,E2 -5522.519} C_VEL
LIN {X 0,Y 509.833,Z 341.604,A -85,B 0,C 180,E1 -5525.58,E2 -5525.58} C_VEL
LIN {X 0,Y 509.851,Z 341.602,A -85,B 0,C 180,E1 -5528.338,E2 -5528.338} C_VEL
LIN {X 0,Y 509.856,Z 341.599,A -85,B 0,C 180,E1 -5531.426,E2 -5531.426} C_VEL
LIN {X 0,Y 509.84,Z 341.606,A -85,B 0,C 180,E1 -5534.67,E2 -5534.67} C_VEL
LIN {X 0,Y 509.851,Z 341.602,A -85,B 0,C 180,E1 -5538.104,E2 -5538.104} C_VEL
LIN {X 0,Y 509.846,Z 341.604,A -85,B 0,C 180,E1 -5540.648,E2 -5540.648} C_VEL
LIN {X 0,Y 509.809,Z 341.605,A -85,B 0,C 180,E1 -5543.646,E2 -5543.646} C_VEL
LIN {X 0,Y 509.848,Z 341.605,A -85,B 0,C 180,E1 -5546.538,E2 -5546.538} C_VEL
LIN {X 0,Y 509.834,Z 341.604,A -85,B 0,C 180,E1 -5549.334,E2 -5549.334} C_VEL
LIN {X 0,Y 509.85,Z 341.783,A -85,B 0,C 180,E1 -5552.415,E2 -5552.415} C_VEL
LIN {X 0,Y 512.629,Z 353.106,A -85,B 0,C 180,E1 -5554.415,E2 -5554.415} C_VEL
LIN {X 0,Y 513.223,Z 357.291,A -85,B 0,C 180,E1 -5555.097,E2 -5555.097} C_VEL
LIN {X 0,Y 512.206,Z 380.065,A -85,B 0,C 180,E1 -5558.467,E2 -5558.467} C_VEL
LIN {X 0,Y 511.591,Z 397.902,A -85,B 0,C 180,E1 -5561.006,E2 -5561.006} C_VEL
LIN {X 0,Y 513.996,Z 410.861,A -85,B 0,C 180,E1 -5561.348,E2 -5561.348} C_VEL
LIN {X 0,Y 512.919,Z 512.766,A -85,B 0,C 180,E1 -5562.944,E2 -5562.944} C_VEL
LIN {X 0,Y 512.644,Z 539.223,A -85,B 0,C 180,E1 -5563.38,E2 -5563.38} C_VEL
LIN {X 0,Y 512.377,Z 553.906,A -85,B 0,C 180,E1 -5563.789,E2 -5563.789} C_VEL
LIN {X 0,Y 512.074,Z 567.349,A -85,B 0,C 180,E1 -5564.324,E2 -5564.324} C_VEL
LIN {X 0,Y 511.716,Z 579.912,A -85,B 0,C 180,E1 -5564.976,E2 -5564.976} C_VEL
LIN {X 0,Y 511.268,Z 592.241,A -85,B 0,C 180,E1 -5565.776,E2 -5565.776} C_VEL
LIN {X 0,Y 510.897,Z 603.524,A -85,B 0,C 180,E1 -5566.679,E2 -5566.679} C_VEL
LIN {X 0,Y 510.485,Z 613.797,A -85,B 0,C 180,E1 -5567.669,E2 -5567.669} C_VEL
LIN {X 0,Y 510.156,Z 624.162,A -85,B 0,C 180,E1 -5568.88,E2 -5568.88} C_VEL
LIN {X 0,Y 509.861,Z 632.635,A -85,B 0,C 180,E1 -5570.078,E2 -5570.078} C_VEL
LIN {X 0,Y 509.611,Z 640.705,A -85,B 0,C 180,E1 -5571.474,E2 -5571.474} C_VEL
LIN {X 0,Y 509.4,Z 647.189,A -85,B 0,C 180,E1 -5572.867,E2 -5572.867} C_VEL
LIN {X 0,Y 509.378,Z 651.644,A -85,B 0,C 180,E1 -5574.061,E2 -5574.061} C_VEL
LIN {X 0,Y 509.196,Z 655.171,A -85,B 0,C 180,E1 -5575.25,E2 -5575.25} C_VEL
LIN {X 0,Y 509.27,Z 657.074,A -85,B 0,C 180,E1 -5576.043,E2 -5576.043} C_VEL
LIN {X 0,Y 509.188,Z 659.764,A -85,B 0,C 180,E1 -5577.627,E2 -5577.627} C_VEL
LIN {X 0,Y 509.07,Z 661.133,A -85,B 0,C 180,E1 -5579.209,E2 -5579.209} C_VEL
LIN {X 0,Y 509.071,Z 661.143,A -85,B 0,C 180,E1 -5580.791,E2 -5580.791} C_VEL
LIN {X 0,Y 509.188,Z 659.842,A -85,B 0,C 180,E1 -5582.373,E2 -5582.373} C_VEL
LIN {X 0,Y 509.27,Z 657.192,A -85,B 0,C 180,E1 -5583.957,E2 -5583.957} C_VEL
LIN {X 0,Y 509.328,Z 653.076,A -85,B 0,C 180,E1 -5585.543,E2 -5585.543} C_VEL
LIN {X 0,Y 509.381,Z 648.582,A -85,B 0,C 180,E1 -5586.845,E2 -5586.845} C_VEL
LIN {X 0,Y 509.544,Z 642.03,A -85,B 0,C 180,E1 -5588.327,E2 -5588.327} C_VEL
LIN {X 0,Y 509.801,Z 634.287,A -85,B 0,C 180,E1 -5589.723,E2 -5589.723} C_VEL
LIN {X 0,Y 510.131,Z 624.683,A -85,B 0,C 180,E1 -5591.121,E2 -5591.121} C_VEL
LIN {X 0,Y 510.452,Z 614.863,A -85,B 0,C 180,E1 -5592.292,E2 -5592.292} C_VEL
LIN {X 0,Y 510.825,Z 604.424,A -85,B 0,C 180,E1 -5593.324,E2 -5593.324} C_VEL
LIN {X 0,Y 511.276,Z 592.076,A -85,B 0,C 180,E1 -5594.325,E2 -5594.325} C_VEL
LIN {X 0,Y 511.704,Z 579.821,A -85,B 0,C 180,E1 -5595.127,E2 -5595.127} C_VEL
LIN {X 0,Y 512.131,Z 566.195,A -85,B 0,C 180,E1 -5595.828,E2 -5595.828} C_VEL
LIN {X 0,Y 512.461,Z 551.671,A -85,B 0,C 180,E1 -5596.39,E2 -5596.39} C_VEL
LIN {X 0,Y 512.74,Z 536.897,A -85,B 0,C 180,E1 -5596.78,E2 -5596.78} C_VEL
LIN {X 0,Y 513.805,Z 410.688,A -85,B 0,C 180,E1 -5598.691,E2 -5598.691} C_VEL
LIN {X 0,Y 511.398,Z 397.467,A -85,B 0,C 180,E1 -5599.022,E2 -5599.022} C_VEL
LIN {X 0,Y 512.13,Z 375.361,A -85,B 0,C 180,E1 -5602.172,E2 -5602.172} C_VEL
LIN {X 0,Y 512.871,Z 356.426,A -85,B 0,C 180,E1 -5604.921,E2 -5604.921} C_VEL
LIN {X 0,Y 512.245,Z 352.064,A -85,B 0,C 180,E1 -5605.606,E2 -5605.606} C_VEL
LIN {X 0,Y 509.857,Z 341.776,A -85,B 0,C 180,E1 -5607.335,E2 -5607.335} C_VEL
LIN {X 0,Y 509.802,Z 341.607,A -85,B 0,C 180,E1 -5610.669,E2 -5610.669} C_VEL
LIN {X 0,Y 509.815,Z 341.603,A -85,B 0,C 180,E1 -5612.959,E2 -5612.959} C_VEL
LIN {X 0,Y 509.143,Z 341.691,A -85,B 0,C 180,E1 -5613.618,E2 -5613.618} C_VEL
LIN {X 0,Y 506.272,Z 342.047,A -85,B 0,C 180,E1 -5614.688,E2 -5614.688} C_VEL
LIN {X 0,Y 503.842,Z 342.351,A -85,B 0,C 180,E1 -5615.55,E2 -5615.55} C_VEL
LIN {X 0,Y 502.794,Z 342.483,A -85,B 0,C 180,E1 -5616.216,E2 -5616.216} C_VEL
LIN {X 0,Y 502.706,Z 342.489,A -85,B 0,C 180,E1 -5616.441,E2 -5616.441} C_VEL
LIN {X 0,Y 502.768,Z 342.48,A -85,B 0,C 180,E1 -5618.979,E2 -5618.979} C_VEL
LIN {X 0,Y 502.746,Z 342.479,A -85,B 0,C 180,E1 -5622.192,E2 -5622.192} C_VEL
LIN {X 0,Y 502.779,Z 342.48,A -85,B 0,C 180,E1 -5625.471,E2 -5625.471} C_VEL
LIN {X 0,Y 502.75,Z 342.483,A -85,B 0,C 180,E1 -5628.927,E2 -5628.927} C_VEL
LIN {X 0,Y 502.754,Z 342.489,A -85,B 0,C 180,E1 -5632.042,E2 -5632.042} C_VEL
LIN {X 0,Y 502.753,Z 342.482,A -85,B 0,C 180,E1 -5635.03,E2 -5635.03} C_VEL
LIN {X 0,Y 502.756,Z 342.485,A -85,B 0,C 180,E1 -5637.913,E2 -5637.913} C_VEL
LIN {X 0,Y 502.771,Z 342.617,A -85,B 0,C 180,E1 -5640.358,E2 -5640.358} C_VEL
LIN {X 0,Y 506.527,Z 358.074,A -85,B 0,C 180,E1 -5642.622,E2 -5642.622} C_VEL
LIN {X 0,Y 506.476,Z 365.893,A -85,B 0,C 180,E1 -5643.638,E2 -5643.638} C_VEL
LIN {X 0,Y 505.688,Z 388.214,A -85,B 0,C 180,E1 -5646.456,E2 -5646.456} C_VEL
LIN {X 0,Y 505.562,Z 398.155,A -85,B 0,C 180,E1 -5647.641,E2 -5647.641} C_VEL
LIN {X 0,Y 508.734,Z 415.224,A -85,B 0,C 180,E1 -5648.051,E2 -5648.051} C_VEL
LIN {X 0,Y 507.485,Z 564.366,A -85,B 0,C 180,E1 -5650.232,E2 -5650.232} C_VEL
LIN {X 0,Y 507.11,Z 579.798,A -85,B 0,C 180,E1 -5650.608,E2 -5650.608} C_VEL
LIN {X 0,Y 506.647,Z 594.566,A -85,B 0,C 180,E1 -5651.133,E2 -5651.133} C_VEL
LIN {X 0,Y 506.143,Z 608.63,A -85,B 0,C 180,E1 -5651.795,E2 -5651.795} C_VEL
LIN {X 0,Y 505.564,Z 622.352,A -85,B 0,C 180,E1 -5652.61,E2 -5652.61} C_VEL
LIN {X 0,Y 504.883,Z 636.213,A -85,B 0,C 180,E1 -5653.627,E2 -5653.627} C_VEL
LIN {X 0,Y 504.265,Z 648.739,A -85,B 0,C 180,E1 -5654.748,E2 -5654.748} C_VEL
LIN {X 0,Y 503.793,Z 659.254,A -85,B 0,C 180,E1 -5655.87,E2 -5655.87} C_VEL
LIN {X 0,Y 503.3,Z 668.994,A -85,B 0,C 180,E1 -5657.09,E2 -5657.09} C_VEL
LIN {X 0,Y 502.906,Z 678.062,A -85,B 0,C 180,E1 -5658.435,E2 -5658.435} C_VEL
LIN {X 0,Y 502.603,Z 686.473,A -85,B 0,C 180,E1 -5659.933,E2 -5659.933} C_VEL
LIN {X 0,Y 502.375,Z 693.876,A -85,B 0,C 180,E1 -5661.553,E2 -5661.553} C_VEL
LIN {X 0,Y 502.191,Z 699.876,A -85,B 0,C 180,E1 -5663.208,E2 -5663.208} C_VEL
LIN {X 0,Y 502.194,Z 703.227,A -85,B 0,C 180,E1 -5664.378,E2 -5664.378} C_VEL
LIN {X 0,Y 502.095,Z 706.773,A -85,B 0,C 180,E1 -5665.987,E2 -5665.987} C_VEL
LIN {X 0,Y 502.062,Z 709.115,A -85,B 0,C 180,E1 -5667.593,E2 -5667.593} C_VEL
LIN {X 0,Y 501.987,Z 710.309,A -85,B 0,C 180,E1 -5669.198,E2 -5669.198} C_VEL
LIN {X 0,Y 501.988,Z 710.326,A -85,B 0,C 180,E1 -5670.802,E2 -5670.802} C_VEL
LIN {X 0,Y 502.063,Z 709.2,A -85,B 0,C 180,E1 -5672.407,E2 -5672.407} C_VEL
LIN {X 0,Y 502.096,Z 706.929,A -85,B 0,C 180,E1 -5674.013,E2 -5674.013} C_VEL
LIN {X 0,Y 502.192,Z 703.463,A -85,B 0,C 180,E1 -5675.622,E2 -5675.622} C_VEL
LIN {X 0,Y 502.245,Z 698.714,A -85,B 0,C 180,E1 -5677.235,E2 -5677.235} C_VEL
LIN {X 0,Y 502.404,Z 692.553,A -85,B 0,C 180,E1 -5678.852,E2 -5678.852} C_VEL
LIN {X 0,Y 502.727,Z 684.811,A -85,B 0,C 180,E1 -5680.471,E2 -5680.471} C_VEL
LIN {X 0,Y 502.967,Z 676.839,A -85,B 0,C 180,E1 -5681.851,E2 -5681.851} C_VEL
LIN {X 0,Y 503.339,Z 668.176,A -85,B 0,C 180,E1 -5683.114,E2 -5683.114} C_VEL
LIN {X 0,Y 503.931,Z 656.482,A -85,B 0,C 180,E1 -5684.539,E2 -5684.539} C_VEL
LIN {X 0,Y 504.525,Z 645.459,A -85,B 0,C 180,E1 -5685.659,E2 -5685.659} C_VEL
LIN {X 0,Y 505.067,Z 632.234,A -85,B 0,C 180,E1 -5686.782,E2 -5686.782} C_VEL
LIN {X 0,Y 505.747,Z 619.037,A -85,B 0,C 180,E1 -5687.697,E2 -5687.697} C_VEL
LIN {X 0,Y 506.272,Z 605.487,A -85,B 0,C 180,E1 -5688.462,E2 -5688.462} C_VEL
LIN {X 0,Y 506.808,Z 590.151,A -85,B 0,C 180,E1 -5689.136,E2 -5689.136} C_VEL
LIN {X 0,Y 507.28,Z 574.535,A -85,B 0,C 180,E1 -5689.631,E2 -5689.631} C_VEL
LIN {X 0,Y 507.557,Z 558.516,A -85,B 0,C 180,E1 -5689.962,E2 -5689.962} C_VEL
LIN {X 0,Y 508.748,Z 414.924,A -85,B 0,C 180,E1 -5692.043,E2 -5692.043} C_VEL
LIN {X 0,Y 505.535,Z 397.806,A -85,B 0,C 180,E1 -5692.471,E2 -5692.471} C_VEL
LIN {X 0,Y 506.1,Z 375.561,A -85,B 0,C 180,E1 -5695.219,E2 -5695.219} C_VEL
LIN {X 0,Y 506.591,Z 358.672,A -85,B 0,C 180,E1 -5697.392,E2 -5697.392} C_VEL
LIN {X 0,Y 502.805,Z 342.776,A -85,B 0,C 180,E1 -5699.69,E2 -5699.69} C_VEL
LIN {X 0,Y 502.744,Z 342.485,A -85,B 0,C 180,E1 -5699.921,E2 -5699.921} C_VEL
LIN {X 0,Y 502.768,Z 342.48,A -85,B 0,C 180,E1 -5703.036,E2 -5703.036} C_VEL
LIN {X 0,Y 502.737,Z 342.484,A -85,B 0,C 180,E1 -5705.954,E2 -5705.954} C_VEL
LIN {X 0,Y 502.768,Z 342.478,A -85,B 0,C 180,E1 -5708.979,E2 -5708.979} C_VEL
LIN {X 0,Y 502.744,Z 342.485,A -85,B 0,C 180,E1 -5712.192,E2 -5712.192} C_VEL
LIN {X 0,Y 502.785,Z 342.479,A -85,B 0,C 180,E1 -5715.47,E2 -5715.47} C_VEL
LIN {X 0,Y 502.757,Z 342.482,A -85,B 0,C 180,E1 -5718.928,E2 -5718.928} C_VEL
LIN {X 0,Y 502.763,Z 342.486,A -85,B 0,C 180,E1 -5722.043,E2 -5722.043} C_VEL
LIN {X 0,Y 502.787,Z 342.474,A -85,B 0,C 180,E1 -5725.033,E2 -5725.033} C_VEL
LIN {X 0,Y 502.782,Z 342.478,A -85,B 0,C 180,E1 -5727.915,E2 -5727.915} C_VEL
LIN {X 0,Y 502.813,Z 342.474,A -85,B 0,C 180,E1 -5730.711,E2 -5730.711} C_VEL
LIN {X 0,Y 502.774,Z 342.478,A -85,B 0,C 180,E1 -5733.46,E2 -5733.46} C_VEL
LIN {X 0,Y 502.768,Z 342.48,A -85,B 0,C 180,E1 -5736.085,E2 -5736.085} C_VEL
LIN {X 0,Y 502.784,Z 342.473,A -85,B 0,C 180,E1 -5738.689,E2 -5738.689} C_VEL
LIN {X 0,Y 502.823,Z 342.476,A -85,B 0,C 180,E1 -5741.248,E2 -5741.248} C_VEL
LIN {X 0,Y 502.85,Z 342.466,A -85,B 0,C 180,E1 -5744.6,E2 -5744.6} C_VEL
LIN {X 0,Y 502.878,Z 342.461,A -85,B 0,C 180,E1 -5748.039,E2 -5748.039} C_VEL
LIN {X 0,Y 502.864,Z 342.468,A -85,B 0,C 180,E1 -5751.156,E2 -5751.156} C_VEL
LIN {X 0,Y 502.927,Z 342.461,A -85,B 0,C 180,E1 -5753.581,E2 -5753.581} C_VEL
LIN {X 0,Y 502.864,Z 342.464,A -85,B 0,C 180,E1 -5756.795,E2 -5756.795} C_VEL
LIN {X 0,Y 503.033,Z 342.451,A -85,B 0,C 180,E1 -5759.199,E2 -5759.199} C_VEL
LIN {X 0,Y 503.021,Z 342.442,A -85,B 0,C 180,E1 -5762.402,E2 -5762.402} C_VEL
LIN {X 0,Y 502.929,Z 342.461,A -85,B 0,C 180,E1 -5765.613,E2 -5765.613} C_VEL
LIN {X 0,Y 502.868,Z 342.462,A -85,B 0,C 180,E1 -5768.843,E2 -5768.843} C_VEL
LIN {X 0,Y 502.847,Z 342.466,A -85,B 0,C 180,E1 -5772.102,E2 -5772.102} C_VEL
LIN {X 0,Y 502.849,Z 342.473,A -85,B 0,C 180,E1 -5775.4,E2 -5775.4} C_VEL
LIN {X 0,Y 502.827,Z 342.471,A -85,B 0,C 180,E1 -5778.752,E2 -5778.752} C_VEL
LIN {X 0,Y 502.784,Z 342.483,A -85,B 0,C 180,E1 -5781.311,E2 -5781.311} C_VEL
LIN {X 0,Y 502.778,Z 342.475,A -85,B 0,C 180,E1 -5783.914,E2 -5783.914} C_VEL
LIN {X 0,Y 502.865,Z 342.466,A -85,B 0,C 180,E1 -5786.566,E2 -5786.566} C_VEL
LIN {X 0,Y 502.825,Z 342.472,A -85,B 0,C 180,E1 -5789.288,E2 -5789.288} C_VEL
LIN {X 0,Y 502.784,Z 342.478,A -85,B 0,C 180,E1 -5792.084,E2 -5792.084} C_VEL
LIN {X 0,Y 502.799,Z 342.477,A -85,B 0,C 180,E1 -5794.966,E2 -5794.966} C_VEL
LIN {X 0,Y 502.794,Z 342.473,A -85,B 0,C 180,E1 -5797.954,E2 -5797.954} C_VEL
LIN {X 0,Y 502.821,Z 342.462,A -85,B 0,C 180,E1 -5801.066,E2 -5801.066} C_VEL
LIN {X 0,Y 502.801,Z 342.478,A -85,B 0,C 180,E1 -5804.532,E2 -5804.532} C_VEL
LIN {X 0,Y 502.798,Z 342.471,A -85,B 0,C 180,E1 -5807.861,E2 -5807.861} C_VEL
LIN {X 0,Y 502.803,Z 342.483,A -85,B 0,C 180,E1 -5811.024,E2 -5811.024} C_VEL
LIN {X 0,Y 502.775,Z 342.48,A -85,B 0,C 180,E1 -5814.169,E2 -5814.169} C_VEL
LIN {X 0,Y 502.832,Z 342.478,A -85,B 0,C 180,E1 -5816.993,E2 -5816.993} C_VEL
LIN {X 0,Y 502.84,Z 342.479,A -85,B 0,C 180,E1 -5820.508,E2 -5820.508} C_VEL
LIN {X 0,Y 502.917,Z 342.938,A -85,B 0,C 180,E1 -5820.744,E2 -5820.744} C_VEL
LIN {X 0,Y 507.077,Z 358.786,A -85,B 0,C 180,E1 -5823.005,E2 -5823.005} C_VEL
LIN {X 0,Y 507.381,Z 360.576,A -85,B 0,C 180,E1 -5823.245,E2 -5823.245} C_VEL
LIN {X 0,Y 506.206,Z 385.608,A -85,B 0,C 180,E1 -5826.258,E2 -5826.258} C_VEL
LIN {X 0,Y 505.776,Z 397.66,A -85,B 0,C 180,E1 -5827.675,E2 -5827.675} C_VEL
LIN {X 0,Y 506.054,Z 399.939,A -85,B 0,C 180,E1 -5827.771,E2 -5827.771} C_VEL
LIN {X 0,Y 508.394,Z 413.882,A -85,B 0,C 180,E1 -5828.098,E2 -5828.098} C_VEL
LIN {X 0,Y 506.914,Z 564.7,A -85,B 0,C 180,E1 -5830.38,E2 -5830.38} C_VEL
LIN {X 0,Y 506.563,Z 579.912,A -85,B 0,C 180,E1 -5830.766,E2 -5830.766} C_VEL
LIN {X 0,Y 506.193,Z 594.335,A -85,B 0,C 180,E1 -5831.29,E2 -5831.29} C_VEL
LIN {X 0,Y 505.642,Z 608.967,A -85,B 0,C 180,E1 -5831.986,E2 -5831.986} C_VEL
LIN {X 0,Y 505.076,Z 622.545,A -85,B 0,C 180,E1 -5832.801,E2 -5832.801} C_VEL
LIN {X 0,Y 504.519,Z 636.359,A -85,B 0,C 180,E1 -5833.823,E2 -5833.823} C_VEL
LIN {X 0,Y 503.958,Z 648.85,A -85,B 0,C 180,E1 -5834.946,E2 -5834.946} C_VEL
LIN {X 0,Y 503.446,Z 661.057,A -85,B 0,C 180,E1 -5836.272,E2 -5836.272} C_VEL
LIN {X 0,Y 503.079,Z 670.522,A -85,B 0,C 180,E1 -5837.495,E2 -5837.495} C_VEL
LIN {X 0,Y 502.729,Z 679.777,A -85,B 0,C 180,E1 -5838.918,E2 -5838.918} C_VEL
LIN {X 0,Y 502.433,Z 687.442,A -85,B 0,C 180,E1 -5840.337,E2 -5840.337} C_VEL
LIN {X 0,Y 502.291,Z 694.596,A -85,B 0,C 180,E1 -5841.957,E2 -5841.957} C_VEL
LIN {X 0,Y 502.184,Z 700.21,A -85,B 0,C 180,E1 -5843.572,E2 -5843.572} C_VEL
LIN {X 0,Y 502.079,Z 704.445,A -85,B 0,C 180,E1 -5845.182,E2 -5845.182} C_VEL
LIN {X 0,Y 502.105,Z 707.414,A -85,B 0,C 180,E1 -5846.791,E2 -5846.791} C_VEL
LIN {X 0,Y 502.033,Z 709.176,A -85,B 0,C 180,E1 -5848.396,E2 -5848.396} C_VEL
LIN {X 0,Y 501.977,Z 709.77,A -85,B 0,C 180,E1 -5850,E2 -5850} C_VEL
LIN {X 0,Y 502.033,Z 709.153,A -85,B 0,C 180,E1 -5851.604,E2 -5851.604} C_VEL
LIN {X 0,Y 502.105,Z 707.367,A -85,B 0,C 180,E1 -5853.21,E2 -5853.21} C_VEL
LIN {X 0,Y 502.079,Z 704.374,A -85,B 0,C 180,E1 -5854.818,E2 -5854.818} C_VEL
LIN {X 0,Y 502.145,Z 700.107,A -85,B 0,C 180,E1 -5856.429,E2 -5856.429} C_VEL
LIN {X 0,Y 502.291,Z 694.444,A -85,B 0,C 180,E1 -5858.043,E2 -5858.043} C_VEL
LIN {X 0,Y 502.431,Z 687.217,A -85,B 0,C 180,E1 -5859.663,E2 -5859.663} C_VEL
LIN {X 0,Y 502.718,Z 679.466,A -85,B 0,C 180,E1 -5861.083,E2 -5861.083} C_VEL
LIN {X 0,Y 503.047,Z 670.097,A -85,B 0,C 180,E1 -5862.507,E2 -5862.507} C_VEL
LIN {X 0,Y 503.408,Z 660.531,A -85,B 0,C 180,E1 -5863.729,E2 -5863.729} C_VEL
LIN {X 0,Y 503.908,Z 648.177,A -85,B 0,C 180,E1 -5865.056,E2 -5865.056} C_VEL
LIN {X 0,Y 504.49,Z 635.751,A -85,B 0,C 180,E1 -5866.178,E2 -5866.178} C_VEL
LIN {X 0,Y 505.049,Z 621.96,A -85,B 0,C 180,E1 -5867.2,E2 -5867.2} C_VEL
LIN {X 0,Y 505.572,Z 608.326,A -85,B 0,C 180,E1 -5868.017,E2 -5868.017} C_VEL
LIN {X 0,Y 506.117,Z 593.594,A -85,B 0,C 180,E1 -5868.708,E2 -5868.708} C_VEL
LIN {X 0,Y 506.533,Z 578.823,A -85,B 0,C 180,E1 -5869.227,E2 -5869.227} C_VEL
LIN {X 0,Y 506.804,Z 564.825,A -85,B 0,C 180,E1 -5869.572,E2 -5869.572} C_VEL
LIN {X 0,Y 507.908,Z 435.529,A -85,B 0,C 180,E1 -5871.494,E2 -5871.494} C_VEL
LIN {X 0,Y 508.007,Z 412.489,A -85,B 0,C 180,E1 -5871.869,E2 -5871.869} C_VEL
LIN {X 0,Y 505.621,Z 398.064,A -85,B 0,C 180,E1 -5872.231,E2 -5872.231} C_VEL
LIN {X 0,Y 506.668,Z 374.658,A -85,B 0,C 180,E1 -5875.028,E2 -5875.028} C_VEL
LIN {X 0,Y 507.444,Z 360.796,A -85,B 0,C 180,E1 -5876.751,E2 -5876.751} C_VEL
LIN {X 0,Y 504.872,Z 349.837,A -85,B 0,C 180,E1 -5878.372,E2 -5878.372} C_VEL
LIN {X 0,Y 502.853,Z 342.596,A -85,B 0,C 180,E1 -5879.568,E2 -5879.568} C_VEL
LIN {X 0,Y 502.833,Z 342.478,A -85,B 0,C 180,E1 -5883.031,E2 -5883.031} C_VEL
LIN {X 0,Y 502.777,Z 342.482,A -85,B 0,C 180,E1 -5885.951,E2 -5885.951} C_VEL
LIN {X 0,Y 502.802,Z 342.482,A -85,B 0,C 180,E1 -5888.976,E2 -5888.976} C_VEL
LIN {X 0,Y 502.796,Z 342.479,A -85,B 0,C 180,E1 -5892.14,E2 -5892.14} C_VEL
LIN {X 0,Y 502.786,Z 342.48,A -85,B 0,C 180,E1 -5895.47,E2 -5895.47} C_VEL
LIN {X 0,Y 502.795,Z 342.479,A -85,B 0,C 180,E1 -5897.861,E2 -5897.861} C_VEL
LIN {X 0,Y 502.801,Z 342.48,A -85,B 0,C 180,E1 -5901.024,E2 -5901.024} C_VEL
LIN {X 0,Y 502.771,Z 342.486,A -85,B 0,C 180,E1 -5904.17,E2 -5904.17} C_VEL
LIN {X 0,Y 502.833,Z 342.476,A -85,B 0,C 180,E1 -5906.994,E2 -5906.994} C_VEL
LIN {X 0,Y 502.811,Z 342.481,A -85,B 0,C 180,E1 -5910.066,E2 -5910.066} C_VEL
LIN {X 0,Y 502.79,Z 342.599,A -85,B 0,C 180,E1 -5911.99,E2 -5911.99} C_VEL
LIN {X 0,Y 505.581,Z 353.68,A -85,B 0,C 180,E1 -5914.032,E2 -5914.032} C_VEL
LIN {X 0,Y 506.471,Z 359.277,A -85,B 0,C 180,E1 -5914.976,E2 -5914.976} C_VEL
LIN {X 0,Y 505.366,Z 381.856,A -85,B 0,C 180,E1 -5918.376,E2 -5918.376} C_VEL
LIN {X 0,Y 504.746,Z 397.896,A -85,B 0,C 180,E1 -5920.699,E2 -5920.699} C_VEL
LIN {X 0,Y 507.356,Z 411.954,A -85,B 0,C 180,E1 -5921.084,E2 -5921.084} C_VEL
LIN {X 0,Y 506.212,Z 502.412,A -85,B 0,C 180,E1 -5922.555,E2 -5922.555} C_VEL
LIN {X 0,Y 505.821,Z 538.91,A -85,B 0,C 180,E1 -5923.156,E2 -5923.156} C_VEL
LIN {X 0,Y 505.511,Z 553.494,A -85,B 0,C 180,E1 -5923.563,E2 -5923.563} C_VEL
LIN {X 0,Y 505.222,Z 567.108,A -85,B 0,C 180,E1 -5924.106,E2 -5924.106} C_VEL
LIN {X 0,Y 504.829,Z 579.784,A -85,B 0,C 180,E1 -5924.766,E2 -5924.766} C_VEL
LIN {X 0,Y 504.345,Z 592.202,A -85,B 0,C 180,E1 -5925.577,E2 -5925.577} C_VEL
LIN {X 0,Y 503.949,Z 603.559,A -85,B 0,C 180,E1 -5926.491,E2 -5926.491} C_VEL
LIN {X 0,Y 503.512,Z 614.382,A -85,B 0,C 180,E1 -5927.546,E2 -5927.546} C_VEL
LIN {X 0,Y 503.172,Z 624.341,A -85,B 0,C 180,E1 -5928.724,E2 -5928.724} C_VEL
LIN {X 0,Y 502.824,Z 632.86,A -85,B 0,C 180,E1 -5929.938,E2 -5929.938} C_VEL
LIN {X 0,Y 502.563,Z 640.963,A -85,B 0,C 180,E1 -5931.354,E2 -5931.354} C_VEL
LIN {X 0,Y 502.358,Z 647.475,A -85,B 0,C 180,E1 -5932.767,E2 -5932.767} C_VEL
LIN {X 0,Y 502.32,Z 651.97,A -85,B 0,C 180,E1 -5933.977,E2 -5933.977} C_VEL
LIN {X 0,Y 502.118,Z 655.5,A -85,B 0,C 180,E1 -5935.183,E2 -5935.183} C_VEL
LIN {X 0,Y 502.199,Z 657.398,A -85,B 0,C 180,E1 -5935.988,E2 -5935.988} C_VEL
LIN {X 0,Y 502.119,Z 660.111,A -85,B 0,C 180,E1 -5937.594,E2 -5937.594} C_VEL
LIN {X 0,Y 501.987,Z 661.485,A -85,B 0,C 180,E1 -5939.198,E2 -5939.198} C_VEL
LIN {X 0,Y 501.988,Z 661.492,A -85,B 0,C 180,E1 -5940.802,E2 -5940.802} C_VEL
LIN {X 0,Y 502.118,Z 660.173,A -85,B 0,C 180,E1 -5942.407,E2 -5942.407} C_VEL
LIN {X 0,Y 502.198,Z 657.504,A -85,B 0,C 180,E1 -5944.012,E2 -5944.012} C_VEL
LIN {X 0,Y 502.176,Z 654.546,A -85,B 0,C 180,E1 -5945.219,E2 -5945.219} C_VEL
LIN {X 0,Y 502.293,Z 649.93,A -85,B 0,C 180,E1 -5946.649,E2 -5946.649} C_VEL
LIN {X 0,Y 502.433,Z 644.175,A -85,B 0,C 180,E1 -5948.041,E2 -5948.041} C_VEL
LIN {X 0,Y 502.699,Z 636.876,A -85,B 0,C 180,E1 -5949.455,E2 -5949.455} C_VEL
LIN {X 0,Y 503.027,Z 627.809,A -85,B 0,C 180,E1 -5950.872,E2 -5950.872} C_VEL
LIN {X 0,Y 503.331,Z 618.275,A -85,B 0,C 180,E1 -5952.09,E2 -5952.09} C_VEL
LIN {X 0,Y 503.792,Z 607.702,A -85,B 0,C 180,E1 -5953.205,E2 -5953.205} C_VEL
LIN {X 0,Y 504.213,Z 596.014,A -85,B 0,C 180,E1 -5954.221,E2 -5954.221} C_VEL
LIN {X 0,Y 504.755,Z 583.046,A -85,B 0,C 180,E1 -5955.133,E2 -5955.133} C_VEL
LIN {X 0,Y 505.178,Z 569.346,A -85,B 0,C 180,E1 -5955.896,E2 -5955.896} C_VEL
LIN {X 0,Y 505.533,Z 556.322,A -85,B 0,C 180,E1 -5956.449,E2 -5956.449} C_VEL
LIN {X 0,Y 505.873,Z 542.09,A -85,B 0,C 180,E1 -5956.882,E2 -5956.882} C_VEL
LIN {X 0,Y 506.06,Z 527.43,A -85,B 0,C 180,E1 -5957.164,E2 -5957.164} C_VEL
LIN {X 0,Y 507.132,Z 411.634,A -85,B 0,C 180,E1 -5958.943,E2 -5958.943} C_VEL
LIN {X 0,Y 504.544,Z 397.594,A -85,B 0,C 180,E1 -5959.295,E2 -5959.295} C_VEL
LIN {X 0,Y 505.342,Z 375.436,A -85,B 0,C 180,E1 -5962.486,E2 -5962.486} C_VEL
LIN {X 0,Y 506.037,Z 358.193,A -85,B 0,C 180,E1 -5965.024,E2 -5965.024} C_VEL
LIN {X 0,Y 505.686,Z 355.031,A -85,B 0,C 180,E1 -5965.521,E2 -5965.521} C_VEL
LIN {X 0,Y 502.838,Z 342.768,A -85,B 0,C 180,E1 -5967.58,E2 -5967.58} C_VEL
LIN {X 0,Y 502.78,Z 342.482,A -85,B 0,C 180,E1 -5967.922,E2 -5967.922} C_VEL
LIN {X 0,Y 502.763,Z 342.483,A -85,B 0,C 180,E1 -5971.146,E2 -5971.146} C_VEL
LIN {X 0,Y 502.775,Z 342.486,A -85,B 0,C 180,E1 -5973.996,E2 -5973.996} C_VEL
LIN {X 0,Y 502.706,Z 342.489,A -85,B 0,C 180,E1 -5976.441,E2 -5976.441} C_VEL
LIN {X 0,Y 502.034,Z 342.572,A -85,B 0,C 180,E1 -5977.111,E2 -5977.111} C_VEL
LIN {X 0,Y 499.191,Z 342.931,A -85,B 0,C 180,E1 -5978.198,E2 -5978.198} C_VEL
LIN {X 0,Y 496.799,Z 343.227,A -85,B 0,C 180,E1 -5979.075,E2 -5979.075} C_VEL
LIN {X 0,Y 495.783,Z 343.354,A -85,B 0,C 180,E1 -5979.751,E2 -5979.751} C_VEL
LIN {X 0,Y 495.706,Z 343.366,A -85,B 0,C 180,E1 -5979.98,E2 -5979.98} C_VEL
LIN {X 0,Y 495.69,Z 343.354,A -85,B 0,C 180,E1 -5982.887,E2 -5982.887} C_VEL
LIN {X 0,Y 495.713,Z 343.36,A -85,B 0,C 180,E1 -5985.996,E2 -5985.996} C_VEL
LIN {X 0,Y 495.708,Z 343.36,A -85,B 0,C 180,E1 -5989.294,E2 -5989.294} C_VEL
LIN {X 0,Y 495.713,Z 343.358,A -85,B 0,C 180,E1 -5991.405,E2 -5991.405} C_VEL
LIN {X 0,Y 495.715,Z 343.363,A -85,B 0,C 180,E1 -5994.459,E2 -5994.459} C_VEL
LIN {X 0,Y 495.725,Z 343.361,A -85,B 0,C 180,E1 -5997.402,E2 -5997.402} C_VEL
LIN {X 0,Y 495.741,Z 343.516,A -85,B 0,C 180,E1 -6000.077,E2 -6000.077} C_VEL
LIN {X 0,Y 499.585,Z 359.246,A -85,B 0,C 180,E1 -6002.408,E2 -6002.408} C_VEL
LIN {X 0,Y 499.864,Z 362.338,A -85,B 0,C 180,E1 -6002.831,E2 -6002.831} C_VEL
LIN {X 0,Y 499.072,Z 384.488,A -85,B 0,C 180,E1 -6005.675,E2 -6005.675} C_VEL
LIN {X 0,Y 498.736,Z 398.046,A -85,B 0,C 180,E1 -6007.318,E2 -6007.318} C_VEL
LIN {X 0,Y 502.147,Z 416.363,A -85,B 0,C 180,E1 -6007.767,E2 -6007.767} C_VEL
LIN {X 0,Y 500.821,Z 564.221,A -85,B 0,C 180,E1 -6009.958,E2 -6009.958} C_VEL
LIN {X 0,Y 500.391,Z 580.157,A -85,B 0,C 180,E1 -6010.351,E2 -6010.351} C_VEL
LIN {X 0,Y 499.922,Z 594.759,A -85,B 0,C 180,E1 -6010.88,E2 -6010.88} C_VEL
LIN {X 0,Y 499.373,Z 608.584,A -85,B 0,C 180,E1 -6011.539,E2 -6011.539} C_VEL
LIN {X 0,Y 498.772,Z 622.316,A -85,B 0,C 180,E1 -6012.365,E2 -6012.365} C_VEL
LIN {X 0,Y 498.047,Z 636.183,A -85,B 0,C 180,E1 -6013.396,E2 -6013.396} C_VEL
LIN {X 0,Y 497.384,Z 648.714,A -85,B 0,C 180,E1 -6014.532,E2 -6014.532} C_VEL
LIN {X 0,Y 496.865,Z 659.232,A -85,B 0,C 180,E1 -6015.668,E2 -6015.668} C_VEL
LIN {X 0,Y 496.334,Z 668.975,A -85,B 0,C 180,E1 -6016.905,E2 -6016.905} C_VEL
LIN {X 0,Y 495.866,Z 678.283,A -85,B 0,C 180,E1 -6018.309,E2 -6018.309} C_VEL
LIN {X 0,Y 495.551,Z 686.457,A -85,B 0,C 180,E1 -6019.789,E2 -6019.789} C_VEL
LIN {X 0,Y 495.309,Z 693.862,A -85,B 0,C 180,E1 -6021.432,E2 -6021.432} C_VEL
LIN {X 0,Y 495.116,Z 699.74,A -85,B 0,C 180,E1 -6023.07,E2 -6023.07} C_VEL
LIN {X 0,Y 495.104,Z 703.213,A -85,B 0,C 180,E1 -6024.297,E2 -6024.297} C_VEL
LIN {X 0,Y 494.993,Z 706.759,A -85,B 0,C 180,E1 -6025.929,E2 -6025.929} C_VEL
LIN {X 0,Y 494.971,Z 709.102,A -85,B 0,C 180,E1 -6027.559,E2 -6027.559} C_VEL
LIN {X 0,Y 494.907,Z 710.295,A -85,B 0,C 180,E1 -6029.186,E2 -6029.186} C_VEL
LIN {X 0,Y 494.908,Z 710.312,A -85,B 0,C 180,E1 -6030.814,E2 -6030.814} C_VEL
LIN {X 0,Y 494.972,Z 709.186,A -85,B 0,C 180,E1 -6032.441,E2 -6032.441} C_VEL
LIN {X 0,Y 494.993,Z 706.914,A -85,B 0,C 180,E1 -6034.071,E2 -6034.071} C_VEL
LIN {X 0,Y 495.104,Z 703.447,A -85,B 0,C 180,E1 -6035.703,E2 -6035.703} C_VEL
LIN {X 0,Y 495.165,Z 698.696,A -85,B 0,C 180,E1 -6037.339,E2 -6037.339} C_VEL
LIN {X 0,Y 495.328,Z 692.533,A -85,B 0,C 180,E1 -6038.979,E2 -6038.979} C_VEL
LIN {X 0,Y 495.691,Z 684.788,A -85,B 0,C 180,E1 -6040.621,E2 -6040.621} C_VEL
LIN {X 0,Y 495.988,Z 676.178,A -85,B 0,C 180,E1 -6042.12,E2 -6042.12} C_VEL
LIN {X 0,Y 496.47,Z 666.592,A -85,B 0,C 180,E1 -6043.507,E2 -6043.507} C_VEL
LIN {X 0,Y 496.985,Z 656.447,A -85,B 0,C 180,E1 -6044.746,E2 -6044.746} C_VEL
LIN {X 0,Y 497.651,Z 644.656,A -85,B 0,C 180,E1 -6045.953,E2 -6045.953} C_VEL
LIN {X 0,Y 498.24,Z 632.185,A -85,B 0,C 180,E1 -6047.019,E2 -6047.019} C_VEL
LIN {X 0,Y 498.946,Z 618.977,A -85,B 0,C 180,E1 -6047.946,E2 -6047.946} C_VEL
LIN {X 0,Y 499.534,Z 605.414,A -85,B 0,C 180,E1 -6048.72,E2 -6048.72} C_VEL
LIN {X 0,Y 500.067,Z 590.763,A -85,B 0,C 180,E1 -6049.376,E2 -6049.376} C_VEL
LIN {X 0,Y 500.568,Z 575.726,A -85,B 0,C 180,E1 -6049.87,E2 -6049.87} C_VEL
LIN {X 0,Y 500.879,Z 559.921,A -85,B 0,C 180,E1 -6050.213,E2 -6050.213} C_VEL
LIN {X 0,Y 502.118,Z 415.571,A -85,B 0,C 180,E1 -6052.336,E2 -6052.336} C_VEL
LIN {X 0,Y 498.782,Z 398.055,A -85,B 0,C 180,E1 -6052.772,E2 -6052.772} C_VEL
LIN {X 0,Y 498.903,Z 388.553,A -85,B 0,C 180,E1 -6053.906,E2 -6053.906} C_VEL
LIN {X 0,Y 499.709,Z 366.326,A -85,B 0,C 180,E1 -6056.747,E2 -6056.747} C_VEL
LIN {X 0,Y 499.696,Z 359.735,A -85,B 0,C 180,E1 -6057.617,E2 -6057.617} C_VEL
LIN {X 0,Y 496.189,Z 345.327,A -85,B 0,C 180,E1 -6059.718,E2 -6059.718} C_VEL
LIN {X 0,Y 495.716,Z 343.411,A -85,B 0,C 180,E1 -6060.057,E2 -6060.057} C_VEL
LIN {X 0,Y 495.727,Z 343.356,A -85,B 0,C 180,E1 -6063.232,E2 -6063.232} C_VEL
LIN {X 0,Y 495.68,Z 343.362,A -85,B 0,C 180,E1 -6066.082,E2 -6066.082} C_VEL
LIN {X 0,Y 495.728,Z 343.355,A -85,B 0,C 180,E1 -6068.763,E2 -6068.763} C_VEL
LIN {X 0,Y 495.7,Z 343.367,A -85,B 0,C 180,E1 -6071.787,E2 -6071.787} C_VEL
LIN {X 0,Y 495.737,Z 343.355,A -85,B 0,C 180,E1 -6075.141,E2 -6075.141} C_VEL
LIN {X 0,Y 495.721,Z 343.362,A -85,B 0,C 180,E1 -6078.215,E2 -6078.215} C_VEL
LIN {X 0,Y 495.738,Z 343.354,A -85,B 0,C 180,E1 -6081.235,E2 -6081.235} C_VEL
LIN {X 0,Y 495.738,Z 343.352,A -85,B 0,C 180,E1 -6084.461,E2 -6084.461} C_VEL
LIN {X 0,Y 495.752,Z 343.357,A -85,B 0,C 180,E1 -6087.404,E2 -6087.404} C_VEL
LIN {X 0,Y 495.763,Z 343.354,A -85,B 0,C 180,E1 -6090.253,E2 -6090.253} C_VEL
LIN {X 0,Y 495.739,Z 343.352,A -85,B 0,C 180,E1 -6093.27,E2 -6093.27} C_VEL
LIN {X 0,Y 495.74,Z 343.352,A -85,B 0,C 180,E1 -6096.612,E2 -6096.612} C_VEL
LIN {X 0,Y 495.78,Z 343.35,A -85,B 0,C 180,E1 -6099.324,E2 -6099.324} C_VEL
LIN {X 0,Y 495.78,Z 343.35,A -85,B 0,C 180,E1 -6101.828,E2 -6101.828} C_VEL
LIN {X 0,Y 495.79,Z 343.35,A -85,B 0,C 180,E1 -6105.217,E2 -6105.217} C_VEL
LIN {X 0,Y 495.852,Z 343.334,A -85,B 0,C 180,E1 -6108.555,E2 -6108.555} C_VEL
LIN {X 0,Y 495.837,Z 343.346,A -85,B 0,C 180,E1 -6111.851,E2 -6111.851} C_VEL
LIN {X 0,Y 495.893,Z 343.329,A -85,B 0,C 180,E1 -6114.306,E2 -6114.306} C_VEL
LIN {X 0,Y 495.987,Z 343.331,A -85,B 0,C 180,E1 -6117.564,E2 -6117.564} C_VEL
LIN {X 0,Y 495.999,Z 343.319,A -85,B 0,C 180,E1 -6120,E2 -6120} C_VEL
LIN {X 0,Y 495.989,Z 343.318,A -85,B 0,C 180,E1 -6122.436,E2 -6122.436} C_VEL
LIN {X 0,Y 495.885,Z 343.337,A -85,B 0,C 180,E1 -6125.694,E2 -6125.694} C_VEL
LIN {X 0,Y 495.838,Z 343.338,A -85,B 0,C 180,E1 -6128.97,E2 -6128.97} C_VEL
LIN {X 0,Y 495.829,Z 343.341,A -85,B 0,C 180,E1 -6132.035,E2 -6132.035} C_VEL
LIN {X 0,Y 495.825,Z 343.349,A -85,B 0,C 180,E1 -6135.451,E2 -6135.451} C_VEL
LIN {X 0,Y 495.779,Z 343.347,A -85,B 0,C 180,E1 -6138.237,E2 -6138.237} C_VEL
LIN {X 0,Y 495.775,Z 343.347,A -85,B 0,C 180,E1 -6140.756,E2 -6140.756} C_VEL
LIN {X 0,Y 495.744,Z 343.356,A -85,B 0,C 180,E1 -6143.387,E2 -6143.387} C_VEL
LIN {X 0,Y 495.79,Z 343.346,A -85,B 0,C 180,E1 -6146.068,E2 -6146.068} C_VEL
LIN {X 0,Y 495.773,Z 343.354,A -85,B 0,C 180,E1 -6148.815,E2 -6148.815} C_VEL
LIN {X 0,Y 495.756,Z 343.355,A -85,B 0,C 180,E1 -6151.725,E2 -6151.725} C_VEL
LIN {X 0,Y 495.769,Z 343.35,A -85,B 0,C 180,E1 -6154.694,E2 -6154.694} C_VEL
LIN {X 0,Y 495.73,Z 343.355,A -85,B 0,C 180,E1 -6157.562,E2 -6157.562} C_VEL
LIN {X 0,Y 495.767,Z 343.335,A -85,B 0,C 180,E1 -6160.7,E2 -6160.7} C_VEL
LIN {X 0,Y 495.735,Z 343.356,A -85,B 0,C 180,E1 -6164.001,E2 -6164.001} C_VEL
LIN {X 0,Y 495.726,Z 343.348,A -85,B 0,C 180,E1 -6167.117,E2 -6167.117} C_VEL
LIN {X 0,Y 495.76,Z 343.353,A -85,B 0,C 180,E1 -6169.953,E2 -6169.953} C_VEL
LIN {X 0,Y 495.728,Z 343.361,A -85,B 0,C 180,E1 -6172.553,E2 -6172.553} C_VEL
LIN {X 0,Y 495.778,Z 343.355,A -85,B 0,C 180,E1 -6175.457,E2 -6175.457} C_VEL
LIN {X 0,Y 495.755,Z 343.357,A -85,B 0,C 180,E1 -6178.364,E2 -6178.364} C_VEL
LIN {X 0,Y 495.847,Z 343.581,A -85,B 0,C 180,E1 -6180.376,E2 -6180.376} C_VEL
LIN {X 0,Y 500.351,Z 360.846,A -85,B 0,C 180,E1 -6182.886,E2 -6182.886} C_VEL
LIN {X 0,Y 500.54,Z 364.049,A -85,B 0,C 180,E1 -6183.301,E2 -6183.301} C_VEL
LIN {X 0,Y 499.253,Z 390.345,A -85,B 0,C 180,E1 -6186.506,E2 -6186.506} C_VEL
LIN {X 0,Y 498.976,Z 397.954,A -85,B 0,C 180,E1 -6187.397,E2 -6187.397} C_VEL
LIN {X 0,Y 500.625,Z 408.059,A -85,B 0,C 180,E1 -6187.666,E2 -6187.666} C_VEL
LIN {X 0,Y 501.747,Z 415.335,A -85,B 0,C 180,E1 -6187.835,E2 -6187.835} C_VEL
LIN {X 0,Y 500.137,Z 565.276,A -85,B 0,C 180,E1 -6190.157,E2 -6190.157} C_VEL
LIN {X 0,Y 499.761,Z 581.55,A -85,B 0,C 180,E1 -6190.585,E2 -6190.585} C_VEL
LIN {X 0,Y 499.322,Z 595.667,A -85,B 0,C 180,E1 -6191.112,E2 -6191.112} C_VEL
LIN {X 0,Y 498.74,Z 610.29,A -85,B 0,C 180,E1 -6191.834,E2 -6191.834} C_VEL
LIN {X 0,Y 498.159,Z 623.57,A -85,B 0,C 180,E1 -6192.661,E2 -6192.661} C_VEL
LIN {X 0,Y 497.621,Z 635.794,A -85,B 0,C 180,E1 -6193.593,E2 -6193.593} C_VEL
LIN {X 0,Y 497.027,Z 648.237,A -85,B 0,C 180,E1 -6194.731,E2 -6194.731} C_VEL
LIN {X 0,Y 496.457,Z 660.52,A -85,B 0,C 180,E1 -6196.075,E2 -6196.075} C_VEL
LIN {X 0,Y 496.051,Z 670.012,A -85,B 0,C 180,E1 -6197.314,E2 -6197.314} C_VEL
LIN {X 0,Y 495.678,Z 679.311,A -85,B 0,C 180,E1 -6198.758,E2 -6198.758} C_VEL
LIN {X 0,Y 495.354,Z 687.012,A -85,B 0,C 180,E1 -6200.198,E2 -6200.198} C_VEL
LIN {X 0,Y 495.223,Z 694.199,A -85,B 0,C 180,E1 -6201.841,E2 -6201.841} C_VEL
LIN {X 0,Y 495.086,Z 700.076,A -85,B 0,C 180,E1 -6203.557,E2 -6203.557} C_VEL
LIN {X 0,Y 495.002,Z 704.091,A -85,B 0,C 180,E1 -6205.113,E2 -6205.113} C_VEL
LIN {X 0,Y 495.025,Z 707.072,A -85,B 0,C 180,E1 -6206.745,E2 -6206.745} C_VEL
LIN {X 0,Y 494.96,Z 708.841,A -85,B 0,C 180,E1 -6208.373,E2 -6208.373} C_VEL
LIN {X 0,Y 494.895,Z 709.433,A -85,B 0,C 180,E1 -6210,E2 -6210} C_VEL
LIN {X 0,Y 494.96,Z 708.811,A -85,B 0,C 180,E1 -6211.627,E2 -6211.627} C_VEL
LIN {X 0,Y 495.025,Z 707.011,A -85,B 0,C 180,E1 -6213.256,E2 -6213.256} C_VEL
LIN {X 0,Y 495.002,Z 703.995,A -85,B 0,C 180,E1 -6214.887,E2 -6214.887} C_VEL
LIN {X 0,Y 495.077,Z 699.695,A -85,B 0,C 180,E1 -6216.521,E2 -6216.521} C_VEL
LIN {X 0,Y 495.223,Z 693.99,A -85,B 0,C 180,E1 -6218.159,E2 -6218.159} C_VEL
LIN {X 0,Y 495.351,Z 686.714,A -85,B 0,C 180,E1 -6219.803,E2 -6219.803} C_VEL
LIN {X 0,Y 495.672,Z 678.907,A -85,B 0,C 180,E1 -6221.242,E2 -6221.242} C_VEL
LIN {X 0,Y 496.038,Z 669.683,A -85,B 0,C 180,E1 -6222.686,E2 -6222.686} C_VEL
LIN {X 0,Y 496.442,Z 660.349,A -85,B 0,C 180,E1 -6223.926,E2 -6223.926} C_VEL
LIN {X 0,Y 496.936,Z 649.234,A -85,B 0,C 180,E1 -6225.167,E2 -6225.167} C_VEL
LIN {X 0,Y 497.568,Z 637.401,A -85,B 0,C 180,E1 -6226.27,E2 -6226.27} C_VEL
LIN {X 0,Y 498.109,Z 624.998,A -85,B 0,C 180,E1 -6227.235,E2 -6227.235} C_VEL
LIN {X 0,Y 498.706,Z 612.057,A -85,B 0,C 180,E1 -6228.061,E2 -6228.061} C_VEL
LIN {X 0,Y 499.263,Z 597.91,A -85,B 0,C 180,E1 -6228.784,E2 -6228.784} C_VEL
LIN {X 0,Y 499.72,Z 583.047,A -85,B 0,C 180,E1 -6229.364,E2 -6229.364} C_VEL
LIN {X 0,Y 500.07,Z 568.489,A -85,B 0,C 180,E1 -6229.766,E2 -6229.766} C_VEL
LIN {X 0,Y 500.323,Z 546.785,A -85,B 0,C 180,E1 -6230.13,E2 -6230.13} C_VEL
LIN {X 0,Y 501.386,Z 423.845,A -85,B 0,C 180,E1 -6231.958,E2 -6231.958} C_VEL
LIN {X 0,Y 501.356,Z 413.523,A -85,B 0,C 180,E1 -6232.135,E2 -6232.135} C_VEL
LIN {X 0,Y 498.852,Z 397.949,A -85,B 0,C 180,E1 -6232.549,E2 -6232.549} C_VEL
LIN {X 0,Y 500.107,Z 373.059,A -85,B 0,C 180,E1 -6235.603,E2 -6235.603} C_VEL
LIN {X 0,Y 500.762,Z 362.924,A -85,B 0,C 180,E1 -6236.893,E2 -6236.893} C_VEL
LIN {X 0,Y 498.462,Z 352.885,A -85,B 0,C 180,E1 -6238.415,E2 -6238.415} C_VEL
LIN {X 0,Y 495.8,Z 343.481,A -85,B 0,C 180,E1 -6239.998,E2 -6239.998} C_VEL
LIN {X 0,Y 495.794,Z 343.355,A -85,B 0,C 180,E1 -6243.245,E2 -6243.245} C_VEL
LIN {X 0,Y 495.723,Z 343.361,A -85,B 0,C 180,E1 -6246.089,E2 -6246.089} C_VEL
LIN {X 0,Y 495.764,Z 343.359,A -85,B 0,C 180,E1 -6248.768,E2 -6248.768} C_VEL
LIN {X 0,Y 495.757,Z 343.355,A -85,B 0,C 180,E1 -6251.781,E2 -6251.781} C_VEL
LIN {X 0,Y 495.738,Z 343.359,A -85,B 0,C 180,E1 -6255.141,E2 -6255.141} C_VEL
LIN {X 0,Y 495.751,Z 343.36,A -85,B 0,C 180,E1 -6258.218,E2 -6258.218} C_VEL
LIN {X 0,Y 495.75,Z 343.357,A -85,B 0,C 180,E1 -6261.408,E2 -6261.408} C_VEL
LIN {X 0,Y 495.744,Z 343.362,A -85,B 0,C 180,E1 -6264.462,E2 -6264.462} C_VEL
LIN {X 0,Y 495.768,Z 343.356,A -85,B 0,C 180,E1 -6267.406,E2 -6267.406} C_VEL
LIN {X 0,Y 495.757,Z 343.36,A -85,B 0,C 180,E1 -6270.253,E2 -6270.253} C_VEL
LIN {X 0,Y 495.781,Z 343.587,A -85,B 0,C 180,E1 -6271.602,E2 -6271.602} C_VEL
LIN {X 0,Y 498.556,Z 354.343,A -85,B 0,C 180,E1 -6273.638,E2 -6273.638} C_VEL
LIN {X 0,Y 499.704,Z 360.323,A -85,B 0,C 180,E1 -6274.688,E2 -6274.688} C_VEL
LIN {X 0,Y 498.782,Z 378.049,A -85,B 0,C 180,E1 -6277.421,E2 -6277.421} C_VEL
LIN {X 0,Y 497.931,Z 397.736,A -85,B 0,C 180,E1 -6280.353,E2 -6280.353} C_VEL
LIN {X 0,Y 499.581,Z 406.413,A -85,B 0,C 180,E1 -6280.631,E2 -6280.631} C_VEL
LIN {X 0,Y 500.759,Z 413.519,A -85,B 0,C 180,E1 -6280.816,E2 -6280.816} C_VEL
LIN {X 0,Y 499.354,Z 513.44,A -85,B 0,C 180,E1 -6282.492,E2 -6282.492} C_VEL
LIN {X 0,Y 498.987,Z 539.755,A -85,B 0,C 180,E1 -6282.951,E2 -6282.951} C_VEL
LIN {X 0,Y 498.678,Z 554.278,A -85,B 0,C 180,E1 -6283.369,E2 -6283.369} C_VEL
LIN {X 0,Y 498.345,Z 568.035,A -85,B 0,C 180,E1 -6283.933,E2 -6283.933} C_VEL
LIN {X 0,Y 497.916,Z 581.448,A -85,B 0,C 180,E1 -6284.654,E2 -6284.654} C_VEL
LIN {X 0,Y 497.404,Z 593.603,A -85,B 0,C 180,E1 -6285.475,E2 -6285.475} C_VEL
LIN {X 0,Y 496.92,Z 605.858,A -85,B 0,C 180,E1 -6286.505,E2 -6286.505} C_VEL
LIN {X 0,Y 496.479,Z 616.715,A -85,B 0,C 180,E1 -6287.619,E2 -6287.619} C_VEL
LIN {X 0,Y 496.131,Z 626.008,A -85,B 0,C 180,E1 -6288.768,E2 -6288.768} C_VEL
LIN {X 0,Y 495.797,Z 634.313,A -85,B 0,C 180,E1 -6290,E2 -6290} C_VEL
LIN {X 0,Y 495.507,Z 642.227,A -85,B 0,C 180,E1 -6291.435,E2 -6291.435} C_VEL
LIN {X 0,Y 495.31,Z 647.761,A -85,B 0,C 180,E1 -6292.663,E2 -6292.663} C_VEL
LIN {X 0,Y 495.215,Z 653.536,A -85,B 0,C 180,E1 -6294.299,E2 -6294.299} C_VEL
LIN {X 0,Y 495.043,Z 655.824,A -85,B 0,C 180,E1 -6295.114,E2 -6295.114} C_VEL
LIN {X 0,Y 495.13,Z 657.723,A -85,B 0,C 180,E1 -6295.93,E2 -6295.93} C_VEL
LIN {X 0,Y 495.052,Z 660.458,A -85,B 0,C 180,E1 -6297.559,E2 -6297.559} C_VEL
LIN {X 0,Y 494.908,Z 661.827,A -85,B 0,C 180,E1 -6299.186,E2 -6299.186} C_VEL
LIN {X 0,Y 494.908,Z 661.841,A -85,B 0,C 180,E1 -6300.814,E2 -6300.814} C_VEL
LIN {X 0,Y 495.051,Z 660.505,A -85,B 0,C 180,E1 -6302.441,E2 -6302.441} C_VEL
LIN {X 0,Y 495.129,Z 657.798,A -85,B 0,C 180,E1 -6304.07,E2 -6304.07} C_VEL
LIN {X 0,Y 495.116,Z 654.828,A -85,B 0,C 180,E1 -6305.294,E2 -6305.294} C_VEL
LIN {X 0,Y 495.244,Z 649.533,A -85,B 0,C 180,E1 -6306.928,E2 -6306.928} C_VEL
LIN {X 0,Y 495.406,Z 644.402,A -85,B 0,C 180,E1 -6308.156,E2 -6308.156} C_VEL
LIN {X 0,Y 495.671,Z 637.064,A -85,B 0,C 180,E1 -6309.59,E2 -6309.59} C_VEL
LIN {X 0,Y 495.946,Z 629.361,A -85,B 0,C 180,E1 -6310.822,E2 -6310.822} C_VEL
LIN {X 0,Y 496.326,Z 619.532,A -85,B 0,C 180,E1 -6312.127,E2 -6312.127} C_VEL
LIN {X 0,Y 496.796,Z 608.814,A -85,B 0,C 180,E1 -6313.29,E2 -6313.29} C_VEL
LIN {X 0,Y 497.251,Z 597.296,A -85,B 0,C 180,E1 -6314.32,E2 -6314.32} C_VEL
LIN {X 0,Y 497.8,Z 584.547,A -85,B 0,C 180,E1 -6315.245,E2 -6315.245} C_VEL
LIN {X 0,Y 498.217,Z 572.165,A -85,B 0,C 180,E1 -6315.966,E2 -6315.966} C_VEL
LIN {X 0,Y 498.629,Z 558.691,A -85,B 0,C 180,E1 -6316.576,E2 -6316.576} C_VEL
LIN {X 0,Y 498.968,Z 544.455,A -85,B 0,C 180,E1 -6317.047,E2 -6317.047} C_VEL
LIN {X 0,Y 499.24,Z 530.014,A -85,B 0,C 180,E1 -6317.354,E2 -6317.354} C_VEL
LIN {X 0,Y 500.505,Z 413.429,A -85,B 0,C 180,E1 -6319.187,E2 -6319.187} C_VEL
LIN {X 0,Y 497.674,Z 397.537,A -85,B 0,C 180,E1 -6319.59,E2 -6319.59} C_VEL
LIN {X 0,Y 498.469,Z 376.951,A -85,B 0,C 180,E1 -6322.594,E2 -6322.594} C_VEL
LIN {X 0,Y 499.207,Z 359.389,A -85,B 0,C 180,E1 -6325.213,E2 -6325.213} C_VEL
LIN {X 0,Y 497.447,Z 350.668,A -85,B 0,C 180,E1 -6326.652,E2 -6326.652} C_VEL
LIN {X 0,Y 495.782,Z 343.56,A -85,B 0,C 180,E1 -6327.891,E2 -6327.891} C_VEL
LIN {X 0,Y 495.71,Z 343.363,A -85,B 0,C 180,E1 -6330.69,E2 -6330.69} C_VEL
LIN {X 0,Y 495.724,Z 343.361,A -85,B 0,C 180,E1 -6333.567,E2 -6333.567} C_VEL
LIN {X 0,Y 495.683,Z 343.365,A -85,B 0,C 180,E1 -6336.548,E2 -6336.548} C_VEL
LIN {X 0,Y 495.709,Z 343.362,A -85,B 0,C 180,E1 -6339.643,E2 -6339.643} C_VEL
LIN {X 0,Y 495.706,Z 343.366,A -85,B 0,C 180,E1 -6339.98,E2 -6339.98} C_VEL
LIN {X 0,Y 495.045,Z 343.452,A -85,B 0,C 180,E1 -6340.658,E2 -6340.658} C_VEL
LIN {X 0,Y 492.166,Z 343.803,A -85,B 0,C 180,E1 -6341.758,E2 -6341.758} C_VEL
LIN {X 0,Y 489.742,Z 344.097,A -85,B 0,C 180,E1 -6342.644,E2 -6342.644} C_VEL
LIN {X 0,Y 488.726,Z 344.222,A -85,B 0,C 180,E1 -6343.33,E2 -6343.33} C_VEL
LIN {X 0,Y 488.658,Z 344.232,A -85,B 0,C 180,E1 -6343.562,E2 -6343.562} C_VEL
LIN {X 0,Y 488.665,Z 344.233,A -85,B 0,C 180,E1 -6346.343,E2 -6346.343} C_VEL
LIN {X 0,Y 488.667,Z 344.241,A -85,B 0,C 180,E1 -6349.67,E2 -6349.67} C_VEL
LIN {X 0,Y 488.646,Z 344.237,A -85,B 0,C 180,E1 -6352.838,E2 -6352.838} C_VEL
LIN {X 0,Y 488.703,Z 344.234,A -85,B 0,C 180,E1 -6355.885,E2 -6355.885} C_VEL
LIN {X 0,Y 488.659,Z 344.242,A -85,B 0,C 180,E1 -6358.818,E2 -6358.818} C_VEL
LIN {X 0,Y 488.698,Z 344.452,A -85,B 0,C 180,E1 -6359.794,E2 -6359.794} C_VEL
LIN {X 0,Y 492.645,Z 360.427,A -85,B 0,C 180,E1 -6362.188,E2 -6362.188} C_VEL
LIN {X 0,Y 493.073,Z 364.058,A -85,B 0,C 180,E1 -6362.695,E2 -6362.695} C_VEL
LIN {X 0,Y 492.237,Z 386.055,A -85,B 0,C 180,E1 -6365.54,E2 -6365.54} C_VEL
LIN {X 0,Y 491.903,Z 397.624,A -85,B 0,C 180,E1 -6366.965,E2 -6366.965} C_VEL
LIN {X 0,Y 495.527,Z 416.787,A -85,B 0,C 180,E1 -6367.462,E2 -6367.462} C_VEL
LIN {X 0,Y 494.172,Z 564.085,A -85,B 0,C 180,E1 -6369.676,E2 -6369.676} C_VEL
LIN {X 0,Y 493.767,Z 578.454,A -85,B 0,C 180,E1 -6370.025,E2 -6370.025} C_VEL
LIN {X 0,Y 493.246,Z 593.78,A -85,B 0,C 180,E1 -6370.571,E2 -6370.571} C_VEL
LIN {X 0,Y 492.609,Z 608.537,A -85,B 0,C 180,E1 -6371.276,E2 -6371.276} C_VEL
LIN {X 0,Y 491.976,Z 622.278,A -85,B 0,C 180,E1 -6372.113,E2 -6372.113} C_VEL
LIN {X 0,Y 491.214,Z 636.151,A -85,B 0,C 180,E1 -6373.158,E2 -6373.158} C_VEL
LIN {X 0,Y 490.508,Z 648.688,A -85,B 0,C 180,E1 -6374.309,E2 -6374.309} C_VEL
LIN {X 0,Y 489.928,Z 659.21,A -85,B 0,C 180,E1 -6375.461,E2 -6375.461} C_VEL
LIN {X 0,Y 489.36,Z 668.955,A -85,B 0,C 180,E1 -6376.715,E2 -6376.715} C_VEL
LIN {X 0,Y 488.842,Z 678.515,A -85,B 0,C 180,E1 -6378.182,E2 -6378.182} C_VEL
LIN {X 0,Y 488.528,Z 686.441,A -85,B 0,C 180,E1 -6379.64,E2 -6379.64} C_VEL
LIN {X 0,Y 488.232,Z 693.847,A -85,B 0,C 180,E1 -6381.307,E2 -6381.307} C_VEL
LIN {X 0,Y 488.05,Z 699.726,A -85,B 0,C 180,E1 -6382.969,E2 -6382.969} C_VEL
LIN {X 0,Y 488.017,Z 703.2,A -85,B 0,C 180,E1 -6384.214,E2 -6384.214} C_VEL
LIN {X 0,Y 487.892,Z 706.746,A -85,B 0,C 180,E1 -6385.87,E2 -6385.87} C_VEL
LIN {X 0,Y 487.883,Z 709.089,A -85,B 0,C 180,E1 -6387.523,E2 -6387.523} C_VEL
LIN {X 0,Y 487.83,Z 710.281,A -85,B 0,C 180,E1 -6389.174,E2 -6389.174} C_VEL
LIN {X 0,Y 487.831,Z 710.299,A -85,B 0,C 180,E1 -6390.825,E2 -6390.825} C_VEL
LIN {X 0,Y 487.884,Z 709.171,A -85,B 0,C 180,E1 -6392.477,E2 -6392.477} C_VEL
LIN {X 0,Y 487.892,Z 706.898,A -85,B 0,C 180,E1 -6394.13,E2 -6394.13} C_VEL
LIN {X 0,Y 488.018,Z 703.43,A -85,B 0,C 180,E1 -6395.786,E2 -6395.786} C_VEL
LIN {X 0,Y 488.091,Z 698.677,A -85,B 0,C 180,E1 -6397.446,E2 -6397.446} C_VEL
LIN {X 0,Y 488.266,Z 692.512,A -85,B 0,C 180,E1 -6399.11,E2 -6399.11} C_VEL
LIN {X 0,Y 488.64,Z 684.764,A -85,B 0,C 180,E1 -6400.776,E2 -6400.776} C_VEL
LIN {X 0,Y 488.963,Z 676.705,A -85,B 0,C 180,E1 -6402.209,E2 -6402.209} C_VEL
LIN {X 0,Y 489.411,Z 668.118,A -85,B 0,C 180,E1 -6403.494,E2 -6403.494} C_VEL
LIN {X 0,Y 490.053,Z 656.411,A -85,B 0,C 180,E1 -6404.96,E2 -6404.96} C_VEL
LIN {X 0,Y 490.785,Z 644.257,A -85,B 0,C 180,E1 -6406.215,E2 -6406.215} C_VEL
LIN {X 0,Y 491.429,Z 632.134,A -85,B 0,C 180,E1 -6407.262,E2 -6407.262} C_VEL
LIN {X 0,Y 492.161,Z 618.915,A -85,B 0,C 180,E1 -6408.202,E2 -6408.202} C_VEL
LIN {X 0,Y 492.777,Z 605.338,A -85,B 0,C 180,E1 -6408.987,E2 -6408.987} C_VEL
LIN {X 0,Y 493.414,Z 590.185,A -85,B 0,C 180,E1 -6409.667,E2 -6409.667} C_VEL
LIN {X 0,Y 493.879,Z 574.759,A -85,B 0,C 180,E1 -6410.172,E2 -6410.172} C_VEL
LIN {X 0,Y 494.227,Z 558.899,A -85,B 0,C 180,E1 -6410.51,E2 -6410.51} C_VEL
LIN {X 0,Y 495.603,Z 417.23,A -85,B 0,C 180,E1 -6412.618,E2 -6412.618} C_VEL
LIN {X 0,Y 491.955,Z 397.895,A -85,B 0,C 180,E1 -6413.108,E2 -6413.108} C_VEL
LIN {X 0,Y 492.323,Z 383.301,A -85,B 0,C 180,E1 -6414.905,E2 -6414.905} C_VEL
LIN {X 0,Y 493.066,Z 363.4,A -85,B 0,C 180,E1 -6417.489,E2 -6417.489} C_VEL
LIN {X 0,Y 491.888,Z 357.335,A -85,B 0,C 180,E1 -6418.364,E2 -6418.364} C_VEL
LIN {X 0,Y 488.684,Z 344.365,A -85,B 0,C 180,E1 -6420.324,E2 -6420.324} C_VEL
LIN {X 0,Y 488.692,Z 344.232,A -85,B 0,C 180,E1 -6423.476,E2 -6423.476} C_VEL
LIN {X 0,Y 488.643,Z 344.239,A -85,B 0,C 180,E1 -6426.348,E2 -6426.348} C_VEL
LIN {X 0,Y 488.668,Z 344.233,A -85,B 0,C 180,E1 -6429.257,E2 -6429.257} C_VEL
LIN {X 0,Y 488.649,Z 344.238,A -85,B 0,C 180,E1 -6432.53,E2 -6432.53} C_VEL
LIN {X 0,Y 488.701,Z 344.232,A -85,B 0,C 180,E1 -6435.197,E2 -6435.197} C_VEL
LIN {X 0,Y 488.658,Z 344.239,A -85,B 0,C 180,E1 -6438.579,E2 -6438.579} C_VEL
LIN {X 0,Y 488.686,Z 344.231,A -85,B 0,C 180,E1 -6440.95,E2 -6440.95} C_VEL
LIN {X 0,Y 488.661,Z 344.238,A -85,B 0,C 180,E1 -6443.866,E2 -6443.866} C_VEL
LIN {X 0,Y 488.702,Z 344.232,A -85,B 0,C 180,E1 -6446.874,E2 -6446.874} C_VEL
LIN {X 0,Y 488.723,Z 344.234,A -85,B 0,C 180,E1 -6449.781,E2 -6449.781} C_VEL
LIN {X 0,Y 488.698,Z 344.227,A -85,B 0,C 180,E1 -6453.078,E2 -6453.078} C_VEL
